(* Init ST08_407_B55_3 Hubtüre 4 Auslauf STN8 AST (ValveSensor) *)
ST08_407_B55_3.sInit.InstName            :='ST08_407_B55_3';
ST08_407_B55_3.sInit.BitName            :='+8_407_B55.3';
ST08_407_B55_3.sInit.Description         :='Hubtüre 4 Auslauf STN8 GST';
ST08_407_B55_3.sInit.SensorType          :=sValveSensorType_INIT;

(* Init ST08_408_B56_0 Rückhaltezylinder links Auslauf STN8 AST (ValveSensor) *)
ST08_408_B56_0.sInit.InstName            :='ST08_408_B56_0';
ST08_408_B56_0.sInit.BitName            :='+8_408_B56.0';
ST08_408_B56_0.sInit.Description         :='Rückhaltezylinder links Auslauf STN8 AST';
ST08_408_B56_0.sInit.SensorType          :=sValveSensorType_WORK;

(* Init ST08_408_B56_1 Rückhaltezylinder links Auslauf STN8 GST (ValveSensor) *)
ST08_408_B56_1.sInit.InstName            :='ST08_408_B56_1';
ST08_408_B56_1.sInit.BitName            :='+8_408_B56.1';
ST08_408_B56_1.sInit.Description         :='Rückhaltezylinder links Auslauf STN8 GST';
ST08_408_B56_1.sInit.SensorType          :=sValveSensorType_INIT;

(* Init ST08_408_B56_2 Rückhaltezylinder rechts Auslauf STN8 AST (ValveSensor) *)
ST08_408_B56_2.sInit.InstName            :='ST08_408_B56_2';
ST08_408_B56_2.sInit.BitName            :='+8_408_B56.2';
ST08_408_B56_2.sInit.Description         :='Rückhaltezylinder rechts Auslauf STN8 AST';
ST08_408_B56_2.sInit.SensorType          :=sValveSensorType_WORK;

(* Init ST08_408_B56_3 Rückhaltezylinder rechts Auslauf STN8 GST (ValveSensor) *)
ST08_408_B56_3.sInit.InstName            :='ST08_408_B56_3';
ST08_408_B56_3.sInit.BitName            :='+8_408_B56.3';
ST08_408_B56_3.sInit.Description         :='Rückhaltezylinder rechts Auslauf STN8 GST';
ST08_408_B56_3.sInit.SensorType          :=sValveSensorType_INIT;

(* Init ST08_408_B56_4 Abstapelzylinder 1 STN8 AST (ValveSensor) *)
ST08_408_B56_4.sInit.InstName            :='ST08_408_B56_4';
ST08_408_B56_4.sInit.BitName            :='+8_408_B56.4';
ST08_408_B56_4.sInit.Description         :='Abstapelzylinder 1 STN8 AST';
ST08_408_B56_4.sInit.SensorType          :=sValveSensorType_WORK;

(* Init ST08_408_B56_5 Abstapelzylinder 1 STN8 GST (ValveSensor) *)
ST08_408_B56_5.sInit.InstName            :='ST08_408_B56_5';
ST08_408_B56_5.sInit.BitName            :='+8_408_B56.5';
ST08_408_B56_5.sInit.Description         :='Abstapelzylinder 1 STN8 GST';
ST08_408_B56_5.sInit.SensorType          :=sValveSensorType_INIT;

(* Init ST08_408_B56_6 Abstapelzylinder 2 STN8 AST (ValveSensor) *)
ST08_408_B56_6.sInit.InstName            :='ST08_408_B56_6';
ST08_408_B56_6.sInit.BitName            :='+8_408_B56.6';
ST08_408_B56_6.sInit.Description         :='Abstapelzylinder 2 STN8 AST';
ST08_408_B56_6.sInit.SensorType          :=sValveSensorType_WORK;

(* Init ST08_408_B56_7 Abstapelzylinder 2 STN8 AST (ValveSensor) *)
ST08_408_B56_7.sInit.InstName            :='ST08_408_B56_7';
ST08_408_B56_7.sInit.BitName            :='+8_408_B56.7';
ST08_408_B56_7.sInit.Description         :='Abstapelzylinder 2 STN8 GST';
ST08_408_B56_7.sInit.SensorType          :=sValveSensorType_INIT;

(*ST08_400_B50_1 Stopper links + rechts Traystapel Auslaufband eingefahren (ValveSensor)*)
ST08_400_B50_1.sInit.InstName            :='ST08_400_B50_1';
ST08_400_B50_1.sInit.BitName            :='+8_400_B50.1';
ST08_400_B50_1.sInit.Description         :='Stopper links + rechts Auslauf STN8 AST';
ST08_400_B50_1.sInit.SensorType          :=sValveSensorType_WORK;

(*ST08_400_B50_2 Stopper links + rechts Traystapel Auslaufband ausgefahren (ValveSensor)*)
ST08_400_B50_2.sInit.InstName            :='ST08_400_B50_2';
ST08_400_B50_2.sInit.BitName            :='+8_400_B50.2';
ST08_400_B50_2.sInit.Description         :='Stopper links + rechts Auslauf STN8 GST';
ST08_400_B50_2.sInit.SensorType          :=sValveSensorType_INIT;

(*ST08_400_B50_3 Stopper links + rechts Traystapel Auslaufband eingefahren (ValveSensor)*)
ST08_400_B50_3.sInit.InstName            :='ST08_400_B50_3';
ST08_400_B50_3.sInit.BitName            :='+8_400_B50.3';
ST08_400_B50_3.sInit.Description         :='Stopper links + rechts Auslauf STN8 AST';
ST08_400_B50_3.sInit.SensorType          :=sValveSensorType_WORK;

(*ST08_400_B50_6 Stopper links + rechts Traystapel Auslaufband ausgefahren (ValveSensor)*)
ST08_400_B50_6.sInit.InstName            :='ST08_400_B50_6';
ST08_400_B50_6.sInit.BitName            :='+8_400_B50.6';
ST08_400_B50_6.sInit.Description         :='Stopper links + rechts Auslauf STN8 GST';
ST08_400_B50_6.sInit.SensorType          :=sValveSensorType_INIT;

(*ST08_401_B50_7 Traystapel schieben hinten ausgefahren (ValveSensor)*)
ST08_401_B50_7.sInit.InstName            :='ST08_401_B50_7';
ST08_401_B50_7.sInit.BitName            :='+8_401_B50.7';
ST08_401_B50_7.sInit.Description         :='Traystapel schieben hinten';
ST08_401_B50_7.sInit.SensorType          :=sValveSensorType_INIT;

(*ST08_412_B58_0 Rüstsatz Förderband Vereinzelner ausgefahren (ValveSensor)*)
ST08_412_B58_0.sInit.InstName            :='ST08_412_B58_0';
ST08_412_B58_0.sInit.BitName          	 :='+8_412_B58.0';
ST08_412_B58_0.sInit.Description         :='Rüstsatz Förderband Vereinzelner STN8 AST';
ST08_412_B58_0.sInit.SensorType          :=sValveSensorType_WORK;

(*ST08_412_B58_1 Rüstsatz Förderband Vereinzelner eingefahren (ValveSensor)*)
ST08_412_B58_1.sInit.InstName            :='ST08_412_B58_1';
ST08_412_B58_1.sInit.BitName          	 :='+8_412_B58.1';
ST08_412_B58_1.sInit.Description         :='Rüstsatz Förderband Vereinzelner STN8 GST';
ST08_412_B58_1.sInit.SensorType          :=sValveSensorType_INIT;

(*ST08_412_B58_2 Rüstsatz Förderband Stopper ausgefahren (ValveSensor)*)
ST08_412_B58_2.sInit.InstName            :='ST08_412_B58_2';
ST08_412_B58_2.sInit.BitName           	 :='+8_412_B58.2';
ST08_412_B58_2.sInit.Description         :='Rüstsatz Förderband Stopper STN8 AST';
ST08_412_B58_2.sInit.SensorType          :=sValveSensorType_WORK;

(*ST08_412_B58_3 Rüstsatz Förderband Stopper eingefahren (ValveSensor)*)
ST08_412_B58_3.sInit.InstName            :='ST08_412_B58_3';
ST08_412_B58_3.sInit.BitName            :='+8_412_B58.3';
ST08_412_B58_3.sInit.Description         :='Rüstsatz Förderband Stopper STN8 GST';
ST08_412_B58_3.sInit.SensorType          :=sValveSensorType_INIT;

(* Init ST08_412_B58_4 Rüstsatz Förderband frei zum Ablegen ISK von SP Maschine Position 1 (DigIn) *)
ST08_412_B58_4.sInit.InstName            :='ST08_412_B58_4';
ST08_412_B58_4.sInit.Description         :='Frei SP Maschine Position 1';
ST08_412_B58_4.sInit.BitInName           :='+8-412_B58.4';
ST08_412_B58_4.sInit.HomePosSignal       :=2; (* 0: Signal=Low, 1: Signal=High, 2: always  *)
ST08_412_B58_4.sInit.MaxTime             :=2000;

(* Init ST08_412_B58_5 Rüstsatz Förderband frei zum Ablegen ISK von SP Maschine Position 2 (DigIn) *)
ST08_412_B58_5.sInit.InstName            :='ST08_412_B58_5';
ST08_412_B58_5.sInit.Description         :='Frei SP Maschine Position 2';
ST08_412_B58_5.sInit.BitInName           :='+8-412_B58.5';
ST08_412_B58_5.sInit.HomePosSignal       :=2; (* 0: Signal=Low, 1: Signal=High, 2: always  *)
ST08_412_B58_5.sInit.MaxTime             :=2000;

(* Init ST08_412_B58_6 Rüstsatz Förderband frei zum Ablegen ISK von SP Maschine Position 3 (DigIn) *)
ST08_412_B58_6.sInit.InstName            :='ST08_412_B58_6';
ST08_412_B58_6.sInit.Description         :='Frei SP Maschine Position 3';
ST08_412_B58_6.sInit.BitInName           :='+8-412_B58.6';
ST08_412_B58_6.sInit.HomePosSignal       :=2; (* 0: Signal=Low, 1: Signal=High, 2: always  *)
ST08_412_B58_6.sInit.MaxTime             :=2000;

(* Init ST08_412_B58_5_35pol Lageerkennung links (DigIn) *)
ST08_412_B58_5_35pol.sInit.InstName            :='ST08_412_B58_5_35pol';
ST08_412_B58_5_35pol.sInit.Description         :=' Lageerkennung rechts';
ST08_412_B58_5_35pol.sInit.BitInName           :='+8-412_B58.5';
ST08_412_B58_5_35pol.sInit.HomePosSignal       :=2; (* 0: Signal=Low, 1: Signal=High, 2: always  *)
ST08_412_B58_5_35pol.sInit.MaxTime             :=2000;

(* Init ST08_412_B58_6_35pol Lageerkennung rechts (DigIn) *)
ST08_412_B58_6_35pol.sInit.InstName            :='ST08_412_B58_6_35pol';
ST08_412_B58_6_35pol.sInit.Description         :=' Lageerkennung links';
ST08_412_B58_6_35pol.sInit.BitInName           :='+8-412_B58.6';
ST08_412_B58_6_35pol.sInit.HomePosSignal    :=2; (* 0: Signal=Low, 1: Signal=High, 2: always  *)
ST08_412_B58_6_35pol.sInit.MaxTime             :=2000;

(* Init ST08_412_B58_7 Rüstsatz Förderband ISK anwesend zum Vereinzeln (DigIn) *)
ST08_412_B58_7.sInit.InstName            :='ST08_412_B58_7';
ST08_412_B58_7.sInit.Description         :='ISK anwesend zum Vereinzeln';
ST08_412_B58_7.sInit.BitInName           :='+8-412_B58.7';
ST08_412_B58_7.sInit.HomePosSignal       :=2; (* 0: Signal=Low, 1: Signal=High, 2: always  *)
ST08_412_B58_7.sInit.MaxTime             :=2000;

(* Init ST08_412_B59_0 Rüstsatz Förderband ISK auf Übergabeposition Roboter Verpackung (DigIn) *)
ST08_412_B59_0.sInit.InstName            :='ST08_412_B59_0';
ST08_412_B59_0.sInit.Description         :='ISK auf Übergabeposition Roboter';
ST08_412_B59_0.sInit.BitInName           :='+8-412_B59.0';
ST08_412_B59_0.sInit.HomePosSignal       :=2; (* 0: Signal=Low, 1: Signal=High, 2: always  *)
ST08_412_B59_0.sInit.MaxTime             :=2000;

(* Init ST08_169_K1 Bandantrieb 1 Einlauf Trays Ein (DigOutIn) *)
ST08_169_K1.sInit.InstName               :='ST08_169_K1';
ST08_169_K1.sInit.Description            :='Bandantrieb 1 Einlauf Trays Ein';
ST08_169_K1.sInit.BitOutName             :='+8-169_K1'; 
ST08_169_K1.sInit.BitInName              :='';
ST08_169_K1.sInit.HomePosOutput          :=2; (* 0: Signal=Low, 1: Signal=High, 2: always  *)
ST08_169_K1.sInit.MaxTime                :=2000;
ST08_169_K1.sInit.EnableInEveryMode  :=TRUE;

(* Init ST08_169_K2 Bandantrieb 4 Auslauf leere Trays Ein (DigOutIn) *)
ST08_169_K2.sInit.InstName               :='ST08_169_K2';
ST08_169_K2.sInit.Description            :='Bandantrieb 4 Auslauf leere Trays Ein';
ST08_169_K2.sInit.BitOutName             :='+8-169_K2'; 
ST08_169_K2.sInit.BitInName              :='';
ST08_169_K2.sInit.HomePosOutput          :=2; (* 0: Signal=Low, 1: Signal=High, 2: always  *)
ST08_169_K2.sInit.MaxTime                :=2000;
ST08_169_K2.sInit.EnableInEveryMode  :=TRUE;

(* Init ST08_170_K1 Bandantrieb 2 Hubquereinheit Trays Ein (DigOutIn) *) 
ST08_170_K1.sInit.InstName               :='ST08_170_K1';
ST08_170_K1.sInit.Description            :='Bandantrieb 2 Hubquereinheit Trays Ein';
ST08_170_K1.sInit.BitOutName             :='+8-170_K1';
ST08_170_K1.sInit.BitInName              :='';
ST08_170_K1.sInit.HomePosOutput          :=2; (* 0: Signal=Low, 1: Signal=High, 2: always  *)
ST08_170_K1.sInit.MaxTime                :=2000;
ST08_170_K1.sInit.EnableInEveryMode  :=TRUE;

(* Init ST08_170_K2 Bandantrieb 3 Hubquereinheit Trays Ein (DigOutIn) *)
ST08_170_K2.sInit.InstName               :='ST08_170_K2';
ST08_170_K2.sInit.Description            :='Bandantrieb 3 Hubquereinheit Trays Ein';
ST08_170_K2.sInit.BitOutName             :='+8-170_K2';
ST08_170_K2.sInit.BitInName              :='';
ST08_170_K2.sInit.HomePosOutput          :=2; (* 0: Signal=Low, 1: Signal=High, 2: always  *)
ST08_170_K2.sInit.MaxTime                :=2000;
ST08_170_K2.sInit.EnableInEveryMode  :=TRUE;

(* Init ST08_400_Y50_0 Stopper Traystapel Einlaufb. hinten links + rechts AST (Valve) *)
ST08_400_Y50_0.sInit.InstName            :='ST08_400_Y50_0';
ST08_400_Y50_0.sInit.BitName            :='+8-400_Y50.0';
ST08_400_Y50_0.sInit.Description         :='Stopper Traystapel Einlaufb. hinten links + rechts AST';
ST08_400_Y50_0.sInit.HomePosDefine       :=HOME_INIT;
ST08_400_Y50_0.sInit.InitDescription     :='GS ausfahren';
ST08_400_Y50_0.sInit.WorkDescription     :='AS einfahren';
ST08_400_Y50_0.sInit.DampBothTime        :=200;
ST08_400_Y50_0.sInit.KindOfValve         :='2G';
ST08_400_Y50_0.sInit.MaxTime             :=2000;

(* Init ST08_400_Y50_2 Stopper Traystapel Einlaufb. mitte links + rechts AST (Valve) *)
ST08_400_Y50_2.sInit.InstName            :='ST08_400_Y50_2';
ST08_400_Y50_2.sInit.BitName            :='+8-400_Y50.2';
ST08_400_Y50_2.sInit.Description         :='Stopper Traystapel Einlaufb. mitte links + rechts AST';
ST08_400_Y50_2.sInit.HomePosDefine       :=HOME_INIT;
ST08_400_Y50_2.sInit.InitDescription     :='GS ausfahren';
ST08_400_Y50_2.sInit.WorkDescription     :='AS einfahren';
ST08_400_Y50_2.sInit.DampBothTime        :=200;
ST08_400_Y50_2.sInit.KindOfValve         :='2G';
ST08_400_Y50_2.sInit.MaxTime             :=2000;

(* Init ST08_402_Y50_4 Stopper Traystapel Einlaufb. vorne links + rechts AST (Valve) *) 
ST08_402_Y50_4.sInit.InstName            :='ST08_402_Y50_4';
ST08_402_Y50_4.sInit.BitName            :='+8-402_Y50.4';
ST08_402_Y50_4.sInit.Description         :='Stopper Traystapel Einlaufb. vorne links + rechts AST';
ST08_402_Y50_4.sInit.HomePosDefine       :=HOME_INIT;
ST08_402_Y50_4.sInit.InitDescription     :='GS ausfahren';
ST08_402_Y50_4.sInit.WorkDescription     :='AS einfahren';
ST08_402_Y50_4.sInit.DampBothTime        :=200;
ST08_402_Y50_4.sInit.KindOfValve         :='2G';
ST08_402_Y50_4.sInit.MaxTime             :=2000;

(* Init ST08_403_Y50_6 Vakuum 1 Einlauf STN8 AST (Valve) *)
ST08_403_Y50_6.sInit.InstName            :='ST08_403_Y50_6';
ST08_403_Y50_6.sInit.BitName            :='+8-403_Y50.6';
ST08_403_Y50_6.sInit.Description         :='Vakuum 1 Einlauf STN8 AST';
ST08_403_Y50_6.sInit.HomePosDefine       :=HOME_ALWAYS;
ST08_403_Y50_6.sInit.InitDescription     :='OFF';
ST08_403_Y50_6.sInit.WorkDescription     :='ON';
ST08_403_Y50_6.sInit.DampBothTime        :=0;
ST08_403_Y50_6.sInit.KindOfValve         :='A';
ST08_403_Y50_6.sInit.MaxTime             :=2000;

(* Init ST08_403_Y50_7 Vakuum 2 Einlauf STN8 AST (Valve) *)
ST08_403_Y50_7.sInit.InstName            :='ST08_403_Y50_7';
ST08_403_Y50_7.sInit.BitName            :='+8-403_Y50.7';
ST08_403_Y50_7.sInit.Description         :='Vakuum 2 Einlauf STN8 AST';
ST08_403_Y50_7.sInit.HomePosDefine       :=HOME_ALWAYS;
ST08_403_Y50_7.sInit.InitDescription     :='OFF';
ST08_403_Y50_7.sInit.WorkDescription     :='ON';
ST08_403_Y50_7.sInit.DampBothTime        :=0;
ST08_403_Y50_7.sInit.KindOfValve         :='A';
ST08_403_Y50_7.sInit.MaxTime             :=2000;

(* Init ST08_405_Y51_0 Hubtüre 2 Einlauf Isokörper STN8 AST (Valve) *)
ST08_405_Y51_0.sInit.InstName            :='ST08_405_Y51_0';
ST08_405_Y51_0.sInit.BitName            :='+8-405_Y51.0';
ST08_405_Y51_0.sInit.Description         :='Hubtüre 2 Einlauf Isokörper STN8 AST';
ST08_405_Y51_0.sInit.HomePosDefine       :=HOME_INIT;
ST08_405_Y51_0.sInit.InitDescription     :='GS ausfahren';
ST08_405_Y51_0.sInit.WorkDescription     :='AS einfahren';
ST08_405_Y51_0.sInit.DampBothTime        :=0;
ST08_405_Y51_0.sInit.KindOfValve         :='2G';
ST08_405_Y51_0.sInit.MaxTime             :=5000;

(* Init ST08_406_Y51_2 Hubtüre 3 STN8 AST (Valve) *)
ST08_406_Y51_2.sInit.InstName            :='ST08_406_Y51_2';
ST08_406_Y51_2.sInit.BitName            :='+8-406_Y51.2';
ST08_406_Y51_2.sInit.Description         :='Hubtüre 3 Auslauf STN8 AST';
ST08_406_Y51_2.sInit.HomePosDefine       :=HOME_INIT;
ST08_406_Y51_2.sInit.InitDescription     :='GS ausfahren';
ST08_406_Y51_2.sInit.WorkDescription     :='AS einfahren';
ST08_406_Y51_2.sInit.DampBothTime        :=0;
ST08_406_Y51_2.sInit.KindOfValve         :='2G';
ST08_406_Y51_2.sInit.MaxTime             :=5000;

(* Init ST08_407_Y51_4 Hubtüre 4 Auslauf STN8 AST (Valve) *)
ST08_407_Y51_4.sInit.InstName            :='ST08_407_Y51_4';
ST08_407_Y51_4.sInit.BitName            :='+8-407_Y51.4';
ST08_407_Y51_4.sInit.Description         :='Hubtüre 4 Auslauf STN8 AST';
ST08_407_Y51_4.sInit.HomePosDefine       :=HOME_ALWAYS;
ST08_407_Y51_4.sInit.InitDescription     :='GS ausfahren';
ST08_407_Y51_4.sInit.WorkDescription     :='AS einfahren';
ST08_407_Y51_4.sInit.DampBothTime        :=0;
ST08_407_Y51_4.sInit.KindOfValve         :='2G';
ST08_407_Y51_4.sInit.MaxTime             :=10000;

(* Init ST08_404_Y51_6 Stopper Traystapel Isokörper AST (Valve) *)
ST08_404_Y51_6.sInit.InstName            :='ST08_404_Y51_6';
ST08_404_Y51_6.sInit.BitName            :='+8-404_Y51.6';
ST08_404_Y51_6.sInit.Description         :='Stopper Traystapel Isokörper AST';
ST08_404_Y51_6.sInit.HomePosDefine       :=HOME_INIT;
ST08_404_Y51_6.sInit.InitDescription     :='GS ausfahren';
ST08_404_Y51_6.sInit.WorkDescription     :='AS einfahren';
ST08_404_Y51_6.sInit.DampBothTime        :=200;
ST08_404_Y51_6.sInit.KindOfValve         :='2G';
ST08_404_Y51_6.sInit.MaxTime             :=2000;

(* Init ST08_404_Y52_0 Hub Bandstrecke STN8 AST (Valve) *)
ST08_404_Y52_0.sInit.InstName            :='ST08_404_Y52_0';
ST08_404_Y52_0.sInit.BitName            :='+8-404_Y52.0';
ST08_404_Y52_0.sInit.Description         :='Hub Bandstrecke STN8 AST';
ST08_404_Y52_0.sInit.HomePosDefine       :=HOME_INIT;
ST08_404_Y52_0.sInit.InitDescription     :='GS einfahren';
ST08_404_Y52_0.sInit.WorkDescription     :='AS ausfahren';
ST08_404_Y52_0.sInit.DampBothTime        :=200;
ST08_404_Y52_0.sInit.KindOfValve         :='2G';
ST08_404_Y52_0.sInit.MaxTime             :=2000;


(* Init ST08_406_Y52_3 Ausheber Trays Entnahmepos. Isok. STN8 GST (Valve) *)
ST08_406_Y52_3.sInit.InstName            :='ST08_406_Y52_3';
ST08_406_Y52_3.sInit.BitName            :='+8-406_Y52.3';
ST08_406_Y52_3.sInit.Description         :='Ausheber Trays Entnahmepos. Isok. STN8 GST';
ST08_406_Y52_3.sInit.HomePosDefine       :=HOME_ALWAYS;
ST08_406_Y52_3.sInit.InitDescription     :='GS einfahren';
ST08_406_Y52_3.sInit.WorkDescription     :='AS ausfahren';
ST08_406_Y52_3.sInit.DampBothTime        :=200;
ST08_406_Y52_3.sInit.KindOfValve         :='2G';
ST08_406_Y52_3.sInit.MaxTime             :=3000;

(* Init ST08_401_Y52_4 Traystapel schieben hinten AST (Valve) *)
ST08_401_Y52_4.sInit.InstName            :='ST08_401_Y52_4';
ST08_401_Y52_4.sInit.BitName            :='+8-401_Y52.4';
ST08_401_Y52_4.sInit.Description         :='Traystapel schieben hinten';
ST08_401_Y52_4.sInit.HomePosDefine       :=HOME_INIT;
ST08_401_Y52_4.sInit.InitDescription     :='GS einfahren';
ST08_401_Y52_4.sInit.WorkDescription     :='AS ausfahren';
ST08_401_Y52_4.sInit.DampBothTime        :=200;
ST08_401_Y52_4.sInit.KindOfValve         :='2G';
ST08_401_Y52_4.sInit.MaxTime             :=2000;

(* Stopper links + rechts Traystapel Auslaufband einfahren (Valve) *)
ST08_400_Y52_5.sInit.InstName            :='ST08_400_Y52_5';
ST08_400_Y52_5.sInit.BitName            :='+8-400_Y52.5';
ST08_400_Y52_5.sInit.Description         :='Stopperzylinder li+re STN8 AST';
ST08_400_Y52_5.sInit.HomePosDefine       :=HOME_BOTH;
ST08_400_Y52_5.sInit.InitDescription     :='GS ausfahren';
ST08_400_Y52_5.sInit.WorkDescription     :='AS einfahren';
ST08_400_Y52_5.sInit.DampBothTime        :=200;
ST08_400_Y52_5.sInit.KindOfValve         :='2G';
ST08_400_Y52_5.sInit.MaxTime             :=3000;

(* Init ST08_402_Y52_6 Traystapel schieben mitte AST (Valve) *)
ST08_402_Y52_6.sInit.InstName            :='ST08_402_Y52_6';
ST08_402_Y52_6.sInit.BitName            :='+8-402_Y52.6';
ST08_402_Y52_6.sInit.Description         :='Traystapel schieben mitte';
ST08_402_Y52_6.sInit.HomePosDefine       :=HOME_INIT;
ST08_402_Y52_6.sInit.InitDescription     :='GS einfahren';
ST08_402_Y52_6.sInit.WorkDescription     :='AS ausfahren';
ST08_402_Y52_6.sInit.DampBothTime        :=200;
ST08_402_Y52_6.sInit.KindOfValve         :='2G';
ST08_402_Y52_6.sInit.MaxTime             :=2000;

(* Init ST08_402_Y52_7 Traystapel schieben vorne AST (Valve) *)
ST08_402_Y52_7.sInit.InstName            :='ST08_402_Y52_7';
ST08_402_Y52_7.sInit.BitName            :='+8-402_Y52.7';
ST08_402_Y52_7.sInit.Description         :='Traystapel schieben vorne';
ST08_402_Y52_7.sInit.HomePosDefine       :=HOME_INIT;
ST08_402_Y52_7.sInit.InitDescription     :='GS einfahren';
ST08_402_Y52_7.sInit.WorkDescription     :='AS ausfahren';
ST08_402_Y52_7.sInit.DampBothTime        :=200;
ST08_402_Y52_7.sInit.KindOfValve         :='2G';
ST08_402_Y52_7.sInit.MaxTime             :=2000;

(* Init ST08_404_Y53_0 Abstapelzylinder 1 AST (Valve) *)
ST08_404_Y53_0.sInit.InstName            :='ST08_404_Y53_0';
ST08_404_Y53_0.sInit.BitName            :='+8-404_Y53.0';
ST08_404_Y53_0.sInit.Description         :='Abstapelzylinder 1 AST';
ST08_404_Y53_0.sInit.HomePosDefine       :=HOME_INIT;
ST08_404_Y53_0.sInit.InitDescription     :='GS einfahren';
ST08_404_Y53_0.sInit.WorkDescription     :='AS ausfahren';
ST08_404_Y53_0.sInit.DampBothTime        :=400;
ST08_404_Y53_0.sInit.KindOfValve         :='2G';
ST08_404_Y53_0.sInit.MaxTime             :=3000;

(* Init ST08_404_Y53_2 Abstapelzylinder 2  AST (Valve) *)
ST08_404_Y53_2.sInit.InstName            :='ST08_404_Y53_2';
ST08_404_Y53_2.sInit.BitName            :='+8-404_Y53.2';
ST08_404_Y53_2.sInit.Description         :='Abstapelzylinder 2  AST';
ST08_404_Y53_2.sInit.HomePosDefine       :=HOME_INIT;
ST08_404_Y53_2.sInit.InitDescription     :='GS einfahren';
ST08_404_Y53_2.sInit.WorkDescription     :='AS ausfahren';
ST08_404_Y53_2.sInit.DampBothTime        :=200;
ST08_404_Y53_2.sInit.KindOfValve         :='2G';
ST08_404_Y53_2.sInit.MaxTime             :=3000;

(* Init ST08_405_Y53_4 Rückhaltezylinder li+re Traystapel Isokörper AST (Valve) *) 
ST08_405_Y53_4.sInit.InstName            :='ST08_405_Y53_4';
ST08_405_Y53_4.sInit.BitName            :='+8-405_Y53.4';
ST08_405_Y53_4.sInit.Description         :='Rückhaltezylinder li+re Traystapel Isokörper AST';
ST08_405_Y53_4.sInit.HomePosDefine       :=HOME_ALWAYS;
ST08_405_Y53_4.sInit.InitDescription     :='GS einfahren';
ST08_405_Y53_4.sInit.WorkDescription     :='AS ausfahren';
ST08_405_Y53_4.sInit.DampBothTime        :=200;
ST08_405_Y53_4.sInit.KindOfValve         :='2G';
ST08_405_Y53_4.sInit.MaxTime             :=3000;

(* Init ST08_408_Y54_0 Rückhaltezylinder li.+re. Auslauf STN8 AST (Valve) *)
ST08_408_Y54_0.sInit.InstName            :='ST08_408_Y54_0';
ST08_408_Y54_0.sInit.BitName            :='+8-408_Y54.0';
ST08_408_Y54_0.sInit.Description         :='Rückhaltezylinder li.+re. Auslauf STN8 AST';
ST08_408_Y54_0.sInit.HomePosDefine       :=HOME_INIT;(*HOME_ALWAYS;*)
ST08_408_Y54_0.sInit.InitDescription     :='GS einfahren';
ST08_408_Y54_0.sInit.WorkDescription     :='AS ausfahren';
ST08_408_Y54_0.sInit.DampBothTime        :=200;
ST08_408_Y54_0.sInit.KindOfValve         :='2G';
ST08_408_Y54_0.sInit.MaxTime             :=3000;

(* Init ST08_408_Y54_2 Abstapelzylinder 1 STN8 AST (Valve) *)
ST08_408_Y54_2.sInit.InstName            :='ST08_408_Y54_2';
ST08_408_Y54_2.sInit.BitName            :='+8-408_Y54.2';
ST08_408_Y54_2.sInit.Description         :='Aufstapelzylinder 1 STN8 AST';
ST08_408_Y54_2.sInit.HomePosDefine       :=HOME_INIT;
ST08_408_Y54_2.sInit.InitDescription     :='GS einfahren';
ST08_408_Y54_2.sInit.WorkDescription     :='AS ausfahren';
ST08_408_Y54_2.sInit.DampBothTime        :=200;
ST08_408_Y54_2.sInit.KindOfValve         :='2G';
ST08_408_Y54_2.sInit.MaxTime             :=3000;

(* Init ST08_408_Y54_4 Abstapelzylinder 2 STN8 AST (Valve) *)
ST08_408_Y54_4.sInit.InstName            :='ST08_408_Y54_4';
ST08_408_Y54_4.sInit.BitName            :='+8-408_Y54.4';
ST08_408_Y54_4.sInit.Description         :='Aufstapelzylinder 2 STN8 AST';
ST08_408_Y54_4.sInit.HomePosDefine       :=HOME_INIT;
ST08_408_Y54_4.sInit.InitDescription     :='GS einfahren';
ST08_408_Y54_4.sInit.WorkDescription     :='AS ausfahren';
ST08_408_Y54_4.sInit.DampBothTime        :=200;
ST08_408_Y54_4.sInit.KindOfValve         :='2G';
ST08_408_Y54_4.sInit.MaxTime             :=3000;

(* Rüstsatz Förderband Vereinzelner (Valve) *)
ST08_412_Y55_0.sInit.InstName            :='ST08_412_Y55_0';
ST08_412_Y55_0.sInit.BitName            :='+8-412_Y55.0';
ST08_412_Y55_0.sInit.Description         :='Rüstsatz Förderband Vereinzelner';
ST08_412_Y55_0.sInit.HomePosDefine       :=HOME_ALWAYS;
ST08_412_Y55_0.sInit.InitDescription     :='GS einfahren';
ST08_412_Y55_0.sInit.WorkDescription     :='AS ausfahren';
ST08_412_Y55_0.sInit.DampBothTime        :=200;
ST08_412_Y55_0.sInit.KindOfValve         :='2G';
ST08_412_Y55_0.sInit.MaxTime             :=3000;

(* Rüstsatz Förderband Stopper (Valve) *)
ST08_412_Y55_2.sInit.InstName            :='ST08_412_Y55_2';
ST08_412_Y55_2.sInit.BitName            :='+8-412_Y55.2';
ST08_412_Y55_2.sInit.Description         :='Rüstsatz Förderband Stopper';
ST08_412_Y55_2.sInit.HomePosDefine       :=HOME_ALWAYS;
ST08_412_Y55_2.sInit.InitDescription     :='GS einfahren';
ST08_412_Y55_2.sInit.WorkDescription     :='AS ausfahren';
ST08_412_Y55_2.sInit.DampBothTime        :=200;
ST08_412_Y55_2.sInit.KindOfValve         :='2G';
ST08_412_Y55_2.sInit.MaxTime             :=3000;
END_PROGRAM

(* POU Stations/ST_03_Ruestsaetze/ST_03_PRGs/ST03_Band_alt, ST *)
PROGRAM ST03_Band_alt
VAR_INPUT
	b_MoveRel 		:BOOL;
	fb_ton_Stopp_Band					: TON;
	bLockBand : BOOL;
END_VAR
VAR
	b_PosBetrieb	:BOOL;
	fb_rTrig_Off		: R_TRIG;
	fb_rTrig_stop		: R_TRIG;
	fb_ton_Off			: TON;
	fb_ton_Off2			: TON;
	fb_rTrig_On			: R_TRIG;
	fb_ton_Stau			: TON;
	fb_ton_Stau2		: TON;
	fb_rtrig_Stopp_Band	: R_TRIG;

	fb_rTrig_MoveRel	: R_TRIG;

	MsgOK				: BOOL;
	MsgCancel			: BOOL;
	lr_PT				: LREAL;
END_VAR
fb_ton_Stopp_Band(IN:= ,PT:=t#10m , Q=> , ET=> );																	(*Stop Wenn von der Sritzguss kein Teile kommen*)

fb_rtrig_Stopp_Band(CLK:=ST00_72_X1_3.BitInToCheck OR ST02_FDB_80_B02.BitInToCheck);
IF	fb_rtrig_Stopp_Band.Q THEN
	fb_ton_Stopp_Band.IN:=FALSE;
END_IF

(*Störung Oriental Motor bei SG-Maschine 3621*)
IF MP.ST03.SGM_3621 THEN
	IF NOT St03_V2.BitInToCheck THEN
		ST03_A5.SetSignalLow := TRUE;

		MessageHandler.Msg.ID:='PM101';
		MessageHandler.Msg.Color:=Color.red;
		MessageHandler.Msg.Name:='Error Förderband';
		MessageHandler.Msg.Text:='Störung Motor Oriental Förderband!';
		MessageHandler.Msg.Station:=3;

		MessageHandler(
			Prio:=2, 							(*1=highest, .. , 4=lowest*)
			Btn1Addr:=ADR(MsgOk),				(*Address of Button1 , if Zero then Button is unvisible*)
			Btn2Addr:=0(*ADR(MsgCancel)*),		(*Address of Button2 , if Zero then Button is unvisible*)
			sVisu:=Visu.Message);
	END_IF
END_IF
(*Motorregelung einschalten=========================================================== *)

IF NOT MP.ST03.SGM_3621 THEN
	IF  NOT ST03_51_M1.Error_ THEN
		IF	(NOT Safety_Fuses_AirPressure.SafetyOK OR gRunEmpty) AND
			ST03_51_M1.on THEN
			ST03_51_M1.MotorOff :=TRUE;
		END_IF

		IF	ModeSelect.Mode > MODE_MANUAL AND
			NOT gRunEmpty AND
			Safety_Fuses_AirPressure.SafetyOK AND
			NOT ST03_51_M1.on THEN
			ST03_51_M1.MotorOn :=TRUE;
		END_IF
	END_IF
END_IF

(*Fahren bis zu Flügelkamera Förderband============================================================ *)

IF	gTypeCode=312  OR		(*93pol*)
	gTypeCode=4991 THEN	(*102pol*)
	b_PosBetrieb:=TRUE;
	(*Impolsbetrieb Förderband============================================================ *)

	IF 	ST03_IFM_Camera.State=STATE_WAIT OR
 		ModeSelect.Mode>=MODE_MANUAL OR
		NOT MP.ST00.IFMCameraActive THEN

		fb_rTrig_MoveRel(CLK:= ST03_51_M1.Ready AND
								b_MoveRel);

		IF	fb_rTrig_MoveRel.Q THEN
			ST03_51_M1.sVelo.maxRpm;
			ST03_51_M1.Vorgabe_Velo:=16000; 			(*mm/min*)
			ST03_51_M1.Vorgabe_Pos_Rel:=MP.ST02.IFMPos;
			ST03_51_M1.MoveRel:=TRUE;
		END_IF

	END_IF

ELSE
	(*Dauerbetrieb Förderband============================================================ *)
	b_PosBetrieb:=FALSE;
	fb_ton_Off(IN:=ST00_73_K3.BitOutToSet , PT:=t#5m, Q=> , ET=> );			(*Stop Wenn von der SG-Maschine keine Teile kommen*)

	IF  gTypeCode = 322 THEN (*160pol*)
		fb_ton_Off2(IN:=ST00_73_K3.BitOutToSet AND								(* Schnittstelle Förderband frei für Spritzmaschine*)
						ST03_422_B64_4.BitInToCheck AND						(* Teil auf Abholposition Roboter *)
						(Robot01.ActualArea<>4), PT:=t#5s , Q=> , ET=> ); 			(*anhalten wenn Roboter nicht in der WT Area ist, die Ablageposition leer und die Abholposition voll ist*)
	ELSE
		fb_ton_Off2(IN:=ST00_73_K3.BitOutToSet AND								(* Schnittstelle Förderband frei für Spritzmaschine*)
						ST08_412_B59_0.BitInToCheck AND						(* Teil auf Abholposition Roboter *)
						(Robot01.ActualArea<>4), PT:=t#3s , Q=> , ET=> ); 		(*anhalten wenn Roboter nicht in der WT Area ist, die Ablageposition leer und die Abholposition voll ist*)
	END_IF

	IF gTypeCode = 5841 THEN	(*268pol*)
		(*Stop wenn 4 Teile auf unterer Führungsschiene belegt sind *)
		fb_ton_Stau2(IN:=	ModeSelect.Mode > MODE_MANUAL AND
							ST03_556_B69_5.BitInToCheck AND	(* Führungsschiene Überwachung Staustrecke*)
							(ST03_556_B69_7. BitInToCheck OR	(* ISK anwesend an Abholposition*)
							Robot01.ActualArea <> 0	AND		(* Roboter zw. Abhol- und Park-Pos.*)
							Robot01.ActualArea <> 5 	AND		(* Blister Pos*)
							Robot01.ActualArea <> 6	), 			(* Park-Pos.*)
							PT:=t#500ms , Q=> , ET=> );
	ELSE
		IF  MP.ST03.SGM_3621 THEN
			fb_ton_Stau.PT:=t#15s;
		ELSE
			lr_PT:=(112-MP.ST02.Override_Band) *0.25;
			fb_ton_Stau.PT:=LREAL_TO_TIME(lr_PT * 1000);
		END_IF
	
		fb_ton_Stau(IN:=	NOT ST00_73_K3.BitOutToSet AND
							Robot01.ActualArea <> 4 AND
							(ModeSelect.Mode = MODE_AUTO_RUN OR ModeSelect.Mode = MODE_AUTO_STOP) ,
							Q=> , ET=>); 			(*Stop wenn Teile nach dem Ablegen nicht weiter gefördert werden*)
	END_IF

	fb_rTrig_Off(CLK:= ModeSelect.Mode<=MODE_MANUAL );

	fb_rTrig_stop(CLK:= ModeSelect.Mode<=MODE_MANUAL AND ST03_51_M1.sVisuAxis.BtnStop.Pressed );

	fb_rTrig_On(CLK:= 	ModeSelect.Mode>MODE_MANUAL AND
						Safety_Fuses_AirPressure.SafetyOK );

	IF NOT MP.ST03.SGM_3621 THEN
		IF	fb_rTrig_On.Q THEN
			ST03_51_M1.MotorOn:=TRUE;
		END_IF

		IF	ST03_51_M1.On THEN
			ST03_51_M1.MoveP:=MP.ST03.BandMoveP;
			ST03_51_M1.MoveN:=NOT MP.ST03.BandMoveP;
		END_IF

		IF 	NOT DummyTest_160pol AND
			(fb_rTrig_Off.Q OR
			fb_ton_Off2.Q OR
			fb_ton_Off.Q OR
			fb_ton_Stau.Q OR
			fb_ton_Stau2.Q OR
			fb_rTrig_stop.Q OR
			bLockBand) THEN
			ST03_51_M1.MotorOn:=FALSE;
			ST03_51_M1.MotorOff:=TRUE;
			ST03_51_M1.MoveN:=FALSE;
			ST03_51_M1.MoveP:=FALSE;
		ELSIF
			DummyTest_160pol AND NOT SpecialMode06.startBand THEN
			ST03_51_M1.MotorOn:=FALSE;
			ST03_51_M1.MotorOff:=TRUE;
			ST03_51_M1.MoveN:=FALSE;
			ST03_51_M1.MoveP:=FALSE;
		END_IF
	ELSE

		(*Ansteuerung Oriental Motor bei SG-Maschine 3621*)

		IF	NOT Safety_Fuses_AirPressure.SafetyOK THEN
			ST03_A5.SetSignalLow:=TRUE;
			ST03_A5.SetSignalHigh :=FALSE;
		ELSIF
			fb_rTrig_Off.Q OR fb_ton_Off2.Q OR fb_ton_Stau.Q THEN
			ST03_A5.SetSignalLow := TRUE;
			ST03_A5.SetSignalHigh :=FALSE;
		ELSIF
			ModeSelect.Mode >MODE_MANUAL AND
			Safety_Fuses_AirPressure.SafetyOK THEN
			ST03_A5.SetSignalHigh :=TRUE;
			ST03_A5.SetSignalLow := FALSE;
		END_IF
	END_IF


END_IF
END_PROGRAM

(* POU zLibrary/ept/Sprache/ST_SwitchLng, ST *)
PROGRAM ST_SwitchLng
VAR_OUTPUT
	b_EndChangeLng		: BOOL;
END_VAR
VAR
	fb_state_entry			: ST_StateEntry;
	s_sprache			: STRING(10);
	b_first_cycle			: BOOL := TRUE;

	btn_Language		: ARRAY [0..3] OF sButtonVisu;

	fbTon_ChangeLng		: TON;
END_VAR
VAR_TEMP
	i					:INT;
END_VAR
fbTon_ChangeLng(
	IN:=	ST_ReadXmlLineMsg.b_EndChangeLng AND
		ST_ReadXmlLine.b_EndChangeLng,
	PT:= t#200ms,
	Q=> b_EndChangeLng,
	ET=> );

IF 	b_first_cycle THEN
	IF	fb_state_entry.fb_ton_Step.ET > t#15s OR
		MP.ST00.Sprache <>'' THEN
		s_sprache := MP.ST00.Sprache;
		CURRENTLANGUAGE:=MP.ST00.Sprache;
		b_first_cycle := FALSE;
	END_IF
ELSE
	MP.ST00.Sprache := CURRENTLANGUAGE;
END_IF
Btn_Init();

IF		btn_Language[1].Pressed THEN
		CURRENTLANGUAGE:= 'DE';
ELSIF
		btn_Language[2].Pressed THEN
		CURRENTLANGUAGE:= 'EN';
ELSIF
		btn_Language[3].Pressed THEN
		CURRENTLANGUAGE:= 'CZ';
END_IF


(* ======================================Schrittkette======================================== *)
fb_state_entry(i16_pos:= 1);

CASE fb_state_entry.i16_step OF
(*=======================================================*)
	INIT_OBJ:

		fb_state_entry.i16_next_step := 10;

(*=======================================================*)
	INIT:
			;

END_CASE

fb_state_entry(i16_pos:= 2 );
END_PROGRAM
ACTION Btn_Init:
btn_Language[1].Text:='DE';
btn_Language[2].Text:='EN';
btn_Language[3].Text:='CZ';

FOR i := 0 TO 3  BY 1DO
	btn_Language[i].Enable:=TRUE;
	btn_Language[i].BackgroundColor:=Color.lightgrey;
	btn_Language[i].TextColor:=Color.black;
	btn_Language[i].Visible:= TRUE;

END_FOR


IF	CURRENTLANGUAGE = 'DE' THEN
	i:=1;
ELSIF
	CURRENTLANGUAGE = 'EN' THEN
	i:=2;
ELSIF
	CURRENTLANGUAGE = 'CZ' THEN
	i:=3;
ELSE
	i:=1;
END_IF

btn_Language[i].BackgroundColor:=Color.grey;
END_ACTION

(* POU zLibrary/ept/Checks/CheckBounds, ST *)
FUNCTION CheckBounds : DINT
VAR_INPUT
	index, lower, upper 	: DINT;
END_VAR
VAR
END_VAR
IF index<lower THEN
	CheckBounds_ErrCnt := CheckBounds_ErrCnt + 1;
	CheckBounds := lower;
ELSIF index>upper THEN
	CheckBounds_ErrCnt := CheckBounds_ErrCnt + 1;
	CheckBounds := upper;
ELSE
	CheckBounds := index;
END_IF
END_FUNCTION

(* POU zLibrary/ept/Checks/CheckDivByte, ST *)
FUNCTION CheckDivByte : BYTE
VAR_INPUT
	divisor			 	: BYTE;
END_VAR
VAR
END_VAR
IF divisor = 0 THEN
	CheckByteZeroDiv_ErrCnt := CheckByteZeroDiv_ErrCnt + 1;
	CheckDivByte := 1;
ELSE
	CheckDivByte := divisor;
END_IF
END_FUNCTION

(* POU zLibrary/ept/Checks/CheckDivDWord, ST *)
FUNCTION CheckDivDWord : DWORD
VAR_INPUT
	divisor				: DWORD;
END_VAR
VAR
END_VAR
IF divisor = 0 THEN
	CheckDWordZeroDiv_ErrCnt := CheckDWordZeroDiv_ErrCnt + 1;
	CheckDivDWord := 1;
ELSE
	CheckDivDWord := divisor;
END_IF
END_FUNCTION

(* POU zLibrary/ept/Checks/CheckDivReal, ST *)
FUNCTION CheckDivReal : REAL
VAR_INPUT
	divisor		 		: REAL;
END_VAR
VAR
END_VAR
IF divisor = 0 THEN
	CheckRealZeroDiv_ErrCnt := CheckRealZeroDiv_ErrCnt + 1;
	CheckDivReal := 1;
ELSE
	CheckDivReal := divisor;
END_IF
END_FUNCTION

(* POU zLibrary/ept/Checks/CheckDivWord, ST *)
FUNCTION CheckDivWord : WORD
VAR_INPUT
	divisor				: WORD;
END_VAR
VAR
END_VAR
IF divisor = 0 THEN
	CheckWordZeroDiv_ErrCnt:= CheckWordZeroDiv_ErrCnt + 1;
	CheckDivWord := 1;
ELSE
	CheckDivWord := divisor;
END_IF
END_FUNCTION

(* POU System/HelpFunctions/CheckProcTime, ST *)
FUNCTION_BLOCK CheckProcTime
VAR_OUTPUT
	PTime		: DINT;	(* Time since start of the timer *)
	Timeout		: BOOL; (* Flag if Timeout occured *)
END_VAR
VAR_INPUT
	MTime		: DINT;	(* Time to timeout *)
	Start		: BOOL;	(* True starts the Timer, False resets *)
END_VAR
VAR
	TONT		: TON;	(* Timer counting Timer *)
END_VAR
(* Start Timer if Start is True.
Stop Timer ,if Start is false.
Timer maximal counting to two hours. *)
TONT(IN:=Start,PT:=T#2h);

(* Updating the Processtime PTime. You get it if you change the output ET of TONT to DWORD.. *)
PTime:=TIME_TO_DWORD(TONT.ET);

(* Setting output Timeout
No Timeout IF Timer stopped OR mtime > ptime*)
IF 	MTime > PTime OR NOT Start THEN
	Timeout:=FALSE;
ELSE
	Timeout:=TRUE;
END_IF
END_FUNCTION_BLOCK

(* POU zLibrary/ept/Checks/CheckRangeSigned, ST *)
FUNCTION CheckRangeSigned : DINT
VAR_INPUT
    value, lower, upper: DINT;
END_VAR
VAR
END_VAR
IF (value < lower) THEN
	CheckRangeSigned_ErrCnt := CheckRangeSigned_ErrCnt + 1;
	CheckRangeSigned := lower;
ELSIF(value > upper) THEN
	CheckRangeSigned_ErrCnt := CheckRangeSigned_ErrCnt + 1;
	CheckRangeSigned := upper;
ELSE
	CheckRangeSigned := value;
END_IF
END_FUNCTION

(* POU zLibrary/ept/Checks/CheckRangeUnsigned, ST *)
FUNCTION CheckRangeUnsigned : UDINT
VAR_INPUT
    value, lower, upper: UDINT;
END_VAR
VAR
END_VAR
IF (value < lower) THEN
	CheckRangeUnSigned_ErrCnt := CheckRangeUnsigned_ErrCnt + 1;
	CheckRangeUnsigned := lower;
ELSIF(value > upper) THEN
	CheckRangeUnsigned_ErrCnt := CheckRangeUnsigned_ErrCnt + 1;
	CheckRangeUnsigned := upper;
ELSE
	CheckRangeUnsigned := value;
END_IF
END_FUNCTION

(* POU zLibrary/ept/Achse/fb_72x1_Achse, ST *)
FUNCTION_BLOCK fb_72x1_Achse   (*Coe-Online 7010.03 (CSV) velocity mode*)
VAR_INPUT
	Stop				:BOOL;			(*aktiven Verfahrbefehl beenden*)
	Reset				:BOOL;			(*Fehler quttieren*)
	MotorOn				:BOOL;			(*Regelung einschalten*)
	MotorOff			:BOOL;			(*Regelung abschalten*)
	NotausOK			:BOOL;
	Override			:DINT;
	Offset				:REAL;			(*  *)
	Vorgabe_Velo		:DINT;			(*in U/min oder mm/min*)
	MoveAbs				:BOOL;			(*startet Positionierung absolut*)
	MoveRel				:BOOL;			(*startet Positionierung relativ*)
	Vorgabe_Pos_Abs		:LREAL:=0;		(*auf diese Position wird bei start MoveAbs gefahren (mm oder Grad)*)
	Vorgabe_Pos_Rel		:LREAL:=0;		(*um diesen Wert wird die Achse bei start MoveRel gefahren (mm oder Grad)*)
	MoveP				:BOOL;			(*Achse bewegt sich in positiver Richtung solange MoveP TRUE ist, oder bis zum Softwarelimit*)
	MoveN				:BOOL;			(*Achse bewegt sich in negativer Richtung solange MoveN TRUE ist, oder bis zum Softwarelimit*)
	bMove				:BOOL;
	sConfig				:st_config_axis;	(*Initialisierung der Achse*)
	sPosList			:ARRAY [1..NO_OF_POS_AXIS] OF st_Pos;

	e_Position			AT %I* :UDINT;
	e_Statusword		AT %I* :UINT;
	e_Velocity			AT %I* :DINT;
	e_Torque			AT %I* :INT;
	e_Following_Error	AT %I* :DINT; 	(*Schleppfehler*)
	e_Toggle			AT %I* :BOOL;
	e_State				AT %I* :UINT;

END_VAR
VAR_OUTPUT
	a_Controlword		AT %Q* :UINT;
	a_Target_Velocity	AT %Q*: DINT;
	a_Target_Position	AT %Q* :UDINT;
	Torque				:ARRAY [1..NO_OF_Torque] OF INT;

	Busy				:BOOL;
	Done				:BOOL;		(*Achse steht auf Position*)
	Error_				:BOOL;
	Ready				:BOOL;
	On					:BOOL;		(*Motor in Regelung*)
	On_Position			:BOOL;		(*Achse steht auf Position*)
	Connect				:BOOL;		(*KLemme ist mit PLC verbunden*)
END_VAR
VAR_IN_OUT
	sVisu				:sDigInVisu;
END_VAR
VAR
	sHelp				:st_Help_axis;
	fb_state_entry		:ST_StateEntry;

	sFb					:st_fb_axis;

	sSm					:st_sm_axis;		(*Störmeldungen*)
	sSmEmpty			:st_sm_axis;
	sCtrl				:st_ctrl_Axis;		(*Control und Status*)
	sCtrlEmpty			:st_ctrl_Axis;

	sVisuAxis			:st_Visu_axis;		(*Taster der Visu*)
	sSdo				:st_sdo;

	(*Variablen für Behr Meldungen*)
	TempErrorText		:STRING(255);
	ProcessTime			:DINT;				(* Counts the time in steps of 100ms since starting operation *)
	Error				:ErrorStruct;
	LaufschriftErrh		:FB_Laufschrift;
	LaufschriftObj		:FB_Laufschrift;

	(*Regler*)
	sVelo				:st_Velo_axis;		(*Geschwindigkeiten*)
	sRegler				:st_PID_axis;		(*Var zur ermittling der Ausgabegeschwindigkeit*)
	sPos				:st_Pos_axis;		(*Positionen*)

	FB_ReadXmlLineConf	:FB_ReadXmlLine;
	FB_ReadXmlLineMsg	:FB_ReadXmlLine;

END_VAR
VAR_TEMP
	i					:INT;
END_VAR

VAR CONSTANT
	NO_OF_Torque		: INT :=50;
END_VAR
(*======================================================
   FB: fb_72x1_Achse (Achse ohne NC verfahren)
 ------------------------------------------------------
   Auth: 		Werner Friedl    						 
   Date: 		18.04.2018   						     
   Rev.: 		1.0	
   Desc:		siehe Aktion " Description "
 ========================================================*)
sub_connect();
sub_Visu();
IF 	NOT sHelp.b_init AND
	sConfig.Aktiv AND
	e_Position<> 0 AND
	Connect  THEN
	sHelp.b_init:=TRUE;
	sPos.r_18bit:=EXPT(2,18);		(*262144 für e_Velocity *)
	sPos.r_20bit:=EXPT(2,20);		(*1048576 für e_Position*)
	sPos.r_32bit:=EXPT(2,32);		(*4294967295 für Überlauf*)
	sConfig.UeberlaufControl_on:=sConfig.SW_Limit_on;
END_IF

IF	sConfig.Aktiv AND
	sConfig.Skalierfaktor <> 0 AND
	sConfig.Getriebefaktor <>0  AND
	sHelp.b_init AND
	Connect THEN
	sub_Regler();
	sub_Pos();
	sub_rec_Torque();
END_IF

Btn_init();
sub_ctrl();
sub_sdo();
sub_fb();

(* Toplevel *)
IF 	fb_state_entry.i16_next_step > INIT AND fb_state_entry.i16_next_step < FEHLER THEN
	IF 	sFb.ton_uez.Q AND NOT sCtrl.in.Fault THEN
		sSm.sm_timeout:=TRUE;
		fb_state_entry.i16_next_step := FEHLER;

	ELSIF
		sCtrl.in.Warning AND NotausOK THEN
		sSm.sm_Error_Warnung:=TRUE;
		fb_state_entry.i16_next_step := FEHLER;

	ELSIF
		fb_state_entry.i16_next_step >= BEREIT AND
		sCtrl.in.Fault THEN
		sSm.sm_Error_Klemme:=TRUE;
		fb_state_entry.i16_next_step := FEHLER;

	ELSIF
		fb_state_entry.i16_next_step >= BEREIT AND
		NOT Connect THEN
		sSm.sm_connect:=TRUE;
		fb_state_entry.i16_next_step := FEHLER;

	ELSIF
		sConfig.ModeOfOperation = CSV AND
		sFb.ton_uez_velo.Q THEN
		sSm.sm_Check_Velo:=TRUE;
	(*	stop:=TRUE;*)

(*	ELSIF fb_state_entry.i16_next_step >= BEREIT AND  sConfig.UeberlaufControl_on AND
		sPos.i32_count_ueberlauf <> 0 THEN
		sSm.sm_Ueberlauf:=TRUE;
		fb_state_entry.i16_next_step := FEHLER;*)
	ELSIF fb_state_entry.i16_next_step >= BEREIT AND  sConfig.Torque_Limit >0 AND
		sConfig.Torque_Limit > e_Torque THEN
		sSm.sm_Torque_zu_gross:=TRUE;
		fb_state_entry.i16_next_step := FEHLER;

	ELSIF sConfig.ModeOfOperation = CSP AND
		sPos.lr_MaxDiff > sConfig.max_PosDiff AND
		sConfig.PosDiffControl_on THEN
		sSm.sm_PosDiff:=TRUE;
		stop:=TRUE;
	END_IF
END_IF

(* ==================================Schrittkette================================ *)
fb_state_entry(	i16_pos:= 1);

CASE fb_state_entry.i16_step OF
(*=======================================================*)
INIT_OBJ:
	fb_state_entry.i16_next_step := INIT;

(*==========================================================================================================*)
INIT:
	IF	 fb_state_entry.E THEN

		sFb.ton_uez.IN := FALSE;
		sFb.ton_quitt.IN := FALSE;
		Stop:=FALSE;
		Reset:=FALSE;
		Busy:=FALSE;
		Error_:=FALSE;
		Done:=FALSE;
		Ready:=FALSE;
		on:=FALSE;

		sCtrl.out:=sCtrlEmpty.out;

	END_IF

		IF	sConfig.aktiv THEN
			fb_state_entry.i16_next_step := 20;
		ELSE
			fb_state_entry.i16_next_step := INAKTIV;
		END_IF

20:(*Switched_on*)

	IF	fb_state_entry.E THEN
		sCtrl.out.Fault_reset:=TRUE;
		sFb.ton_uez.IN:=TRUE;
	END_IF

	(*-----------------------Weiterschaltbedingungen----------------------------*)

	IF	NOT sCtrl.in.Fault THEN
		fb_state_entry.i16_next_step := BEREIT;
		sCtrl.out.Fault_reset:=FALSE;
	ELSE
		IF	sFb.ton_uez.Q THEN
			fb_state_entry.i16_next_step := FEHLER;
		END_IF
	END_IF

(*==========================================================================================================*)
BEREIT:
	IF	fb_state_entry.E THEN
		sFb.ton_uez.IN:=FALSE;
		Ready:=TRUE;
	END_IF

	IF	(sFb.r_trig_MotorOn.Q OR MotorOn)AND
		NOT on THEN
		IF 	NotausOK THEN
			MotorOn:=FALSE;
			sCtrl.out.Target_Position:=sCtrl.in.Position;
			fb_state_entry.i16_next_step := 110;
		ELSE
			sSm.sm_NotausNok:=TRUE;
			fb_state_entry.i16_next_step := FEHLER;
		END_IF
	END_IF

	CASE	sConfig.ModeOfOperation OF

	CSV:
			;
	CSP:
		(*Positionsübergabe*)

		IF 	on AND
			(*Positive Richtung*)
			 ((sVisuAxis.BtnJogP.Pressed AND sVisuAxis.b_kont) OR MoveP) THEN
			IF	sConfig.SW_Limit_on THEN
				IF	sCtrl.in.Position < sConfig.SW_Limit_max THEN
					sCtrl.out.Target_Position:=sConfig.SW_Limit_max;
				END_IF
			ELSE
				sCtrl.out.Target_Position:=sCtrl.in.Position+10000;
			END_IF
			Busy:=TRUE;
			Done:=FALSE;
		END_IF

		IF 	on AND
			(*Negative Richtung*)
			((sVisuAxis.BtnJogM.Pressed AND sVisuAxis.b_kont) OR MoveN) THEN
			IF	sConfig.SW_Limit_on THEN
				IF	sCtrl.in.Position > sConfig.SW_Limit_min THEN
					sCtrl.out.Target_Position:=sConfig.SW_Limit_min;
				END_IF
			ELSE
				sCtrl.out.Target_Position:=sCtrl.in.Position-10000;
			END_IF
			Busy:=TRUE;
			Done:=FALSE;
		END_IF

		(*Jog beenden*)
		IF	sFb.r_trig_jogP.Q OR sFb.r_trig_jogM.Q OR
			sFb.r_trig_MoveP.Q OR sFb.r_trig_MoveM.Q OR
			sFb.r_trig_stop.Q OR reset OR
			Stop  THEN
			Busy:=FALSE;
			Done:=TRUE;
			MoveP:=FALSE;
			MoveN:=FALSE;
			sCtrl.out.Target_Position:=sCtrl.in.Position;
		END_IF


		(*Positionieren mit Positionsvorgabe Absolut*)
		IF	on  AND
			(sFb.r_trig_MoveAbs.Q OR MoveAbs)THEN
			IF	sConfig.SW_Limit_on THEN
				IF	Vorgabe_Pos_Abs > sConfig.SW_Limit_max THEN
					sCtrl.out.Target_Position:=sConfig.SW_Limit_max;
					sSm.sm_SW_Limit:=TRUE;
				ELSIF	Vorgabe_Pos_Abs < sConfig.SW_Limit_min THEN
					sCtrl.out.Target_Position:=sConfig.SW_Limit_min;
					sSm.sm_SW_Limit:=TRUE;
				ELSE
					sCtrl.out.Target_Position:=Vorgabe_Pos_Abs;
					sSm.sm_SW_Limit:=FALSE;
				END_IF
			ELSE
				sCtrl.out.Target_Position:=Vorgabe_Pos_Abs;
			END_IF
			Busy:=TRUE;
			Done:=FALSE;
			bMove:=TRUE;
		END_IF

		(*Positionieren mit Positionsvorgabe Relativ*)
		IF	on  AND
			MoveRel THEN
			IF	sConfig.SW_Limit_on THEN
				IF	Vorgabe_Pos_Rel+sCtrl.out.Target_Position > sConfig.SW_Limit_max THEN
					sCtrl.out.Target_Position:=sConfig.SW_Limit_max;
					sSm.sm_SW_Limit:=TRUE;
				ELSIF	Vorgabe_Pos_Rel+sCtrl.out.Target_Position < sConfig.SW_Limit_min THEN
					sCtrl.out.Target_Position:=sConfig.SW_Limit_min;
					sSm.sm_SW_Limit:=TRUE;
				ELSE
					sCtrl.out.Target_Position:=sCtrl.out.Target_Position+Vorgabe_Pos_Rel;
					sSm.sm_SW_Limit:=FALSE;
				END_IF
			ELSE
				sCtrl.out.Target_Position:=sCtrl.out.Target_Position+Vorgabe_Pos_Rel;
			END_IF
			Busy:=TRUE;
			Done:=FALSE;
			bMove:=TRUE;
		END_IF
		IF	NOT on  AND
			(MoveAbs OR MoveRel)THEN
			fb_state_entry.i16_next_step := FEHLER;
		END_IF
	END_CASE

	(*Regler abschalten*)
	IF	(sFb.r_trig_reset.Q OR MotorOff OR NOT NotausOK )AND
		on	THEN
		sSm.sm_Move:=bMove;
		fb_state_entry.i16_next_step := 210;
	END_IF

	sFb.ton_Busy(IN:=Busy , PT:= t#50ms, Q=> , ET=> );
	IF	sFb.ton_Busy.Q AND On_Position AND
		fb_state_entry.i16_next_step = fb_state_entry.i16_step THEN
		Busy:=FALSE;
		Done:=TRUE;
		bMove:=FALSE;
		IF	sSm.sm_SW_Limit THEN
			fb_state_entry.i16_next_step := FEHLER;
		END_IF
	END_IF

	MotorOff:=FALSE;
	Stop:=FALSE;
	MoveAbs:=FALSE;
	MoveRel:=FALSE;

	IF	fb_state_entry.X THEN
		sFb.ton_uez.IN:=TRUE;
		Busy:=TRUE;
		Error_:=FALSE;
		Done:=FALSE;
		bMove:=FALSE;
	END_IF

(*==========================================================================================================*)
110:(*Ready_to_switch_on*)

	IF	fb_state_entry.E THEN
		sCtrl.out.Enable_voltage:=TRUE;
		sCtrl.out.Shutdown:=TRUE;
		sSm:=sSmEmpty;
	END_IF

	(*-----------------------Weiterschaltbedingungen----------------------------*)
	IF	sCtrl.in.Ready_to_switch_on THEN
		sCtrl.out.Switch_on:=TRUE;
		fb_state_entry.i16_next_step := 120;
	END_IF

(*=======================================================*)
120:(*Switched_on*)

	IF	fb_state_entry.E THEN
		sCtrl.out.Switch_on:=TRUE;
	END_IF

	(*-----------------------Weiterschaltbedingungen----------------------------*)

	IF	sCtrl.in.Switched_on THEN
		fb_state_entry.i16_next_step := 130;
	END_IF

130:(*Operation_enabled*)

	IF	fb_state_entry.E THEN
		sCtrl.out.Enable_operation:=TRUE;
	END_IF

	(*-----------------------Weiterschaltbedingungen----------------------------*)

	IF	sCtrl.in.Operation_enabled THEN
		fb_state_entry.i16_next_step := BEREIT;
		Busy:=FALSE;
		Error_:=FALSE;
		on:=TRUE;
	END_IF

(*==========================================================================================================*)
210:(*Switch_off*)

	IF	fb_state_entry.E THEN
		sCtrl.out.Target_Position:=sCtrl.in.Position;
		sCtrl.out.Enable_operation:=FALSE;
		sCtrl.out.Switch_on:=FALSE;
		on:=FALSE;
		MoveP:=FALSE;
		MoveN:=FALSE;
		Reset:=FALSE;
	END_IF

	(*-----------------------Weiterschaltbedingungen----------------------------*)

	IF	NOT sCtrl.in.Operation_enabled THEN
			fb_state_entry.i16_next_step := 220;
	END_IF

(*=======================================================*)
220:(*Shutdown*)

	IF	fb_state_entry.E THEN
		sCtrl.out.Shutdown:=FALSE;
	END_IF

	(*-----------------------Weiterschaltbedingungen----------------------------*)

	IF	NOT sCtrl.in.Ready_to_switch_on THEN
		fb_state_entry.i16_next_step := 230;
	END_IF

230:(*disabled_voltage*)

	IF	fb_state_entry.E THEN
			sCtrl.out.Enable_voltage:=FALSE;
	END_IF

	(*-----------------------Weiterschaltbedingungen----------------------------*)

	IF	sCtrl.in.Switch_on_disabled THEN
		sCtrl.out.Target_Position:=sCtrl.in.Position;
		fb_state_entry.i16_next_step := 240;
		Busy:=FALSE;
		Error_:=FALSE;
	END_IF

240:(**)
	IF	sSm.sm_PosDiff OR
		sSm.sm_Check_Velo OR
		sSm.sm_Move THEN
		fb_state_entry.i16_next_step := FEHLER;
	ELSE
		fb_state_entry.i16_next_step := BEREIT;
		sSm:=sSmEmpty;
	END_IF

(*==========================================================================================================*)
FEHLER: (*Fehler*)
	IF	fb_state_entry.E THEN
		Busy:=FALSE;
		Error_:=TRUE;
		Ready:=FALSE;
		on:=FALSE;
		MoveP:=FALSE;
		MoveN:=FALSE;
		sCtrl.out:=sCtrlEmpty.out;

		IF	sSm.sm_timeout THEN
			FB_ReadXmlLineMsg.ID:='sm_timeout';
			Error.No:=1;
		ELSIF	sSm.sm_Error_Klemme THEN
			FB_ReadXmlLineMsg.ID:='sm_Error_Klemme';
			Error.No:=2;
		ELSIF	sSm.sm_Error_Warnung THEN
			FB_ReadXmlLineMsg.ID:='sm_Error_Warnung';
			Error.No:=3;
		ELSIF	sSm.sm_Check_Velo THEN
			FB_ReadXmlLineMsg.ID:='sm_Check_Velo';
			Error.No:=4;
		ELSIF	sSm.sm_SW_Limit THEN
			FB_ReadXmlLineMsg.ID:='sm_SW_Limit';
			Error.No:=5;
		ELSIF		sSm.sm_PosDiff THEN
			FB_ReadXmlLineMsg.ID:='sm_PosDiff';
			Error.No:=6;
		ELSIF		sSm.sm_fehler_daten_schreiben THEN
			FB_ReadXmlLineMsg.ID:='sm_fehler_daten_schreiben';
			Error.No:=7;
		ELSIF		sSm.sm_connect THEN
			FB_ReadXmlLineMsg.ID:='sm_connect';
			Error.No:=8;
		ELSIF		sSm.sm_Ueberlauf THEN
			FB_ReadXmlLineMsg.ID:='sm_Ueberlauf';
			Error.No:=9;
		ELSIF			sSm.sm_Torque_zu_gross THEN
			FB_ReadXmlLineMsg.ID:='sm_Torque_zu_gross';
			Error.No:=10;
		ELSIF
			sSm.sm_NotausNok	THEN
			FB_ReadXmlLineMsg.ID:='sm_NotausNok';
			Error.No:=11;
		ELSIF
			sSm.sm_Move	THEN
			FB_ReadXmlLineMsg.ID:='sm_Move';
			Error.No:=12;
		END_IF

		Error.DateTime:=gVarDTSystemtime;

	END_IF

	sVisu.ProcessTime:=ProcessTime;

	IF	sFb.r_trig_quitt.Q THEN
			fb_state_entry.i16_next_step := INIT;
	END_IF

	IF sFb.ton_quitt.Q THEN
		sFb.ton_quitt(IN := FALSE);
	END_IF

INAKTIV:

	Busy:=FALSE;
	Ready := TRUE;
	Done := TRUE;

	IF	sConfig.aktiv THEN
		fb_state_entry.i16_next_step := FEHLER;
	END_IF

END_CASE

fb_state_entry(i16_pos:= 2);


(*------------------------------------------------------------------
	Error-Handling
  ------------------------------------------------------------------*)
IF	sVisuAxis.BtnReset.Pressed OR Reset THEN
	sSm:=sSmEmpty;
END_IF
IF	(MEMCMP(ADR(sSmEmpty), ADR(sSm), SIZEOF(sSmEmpty)) = 0 ) THEN
	Error.No:=0;
	Error.Text:='';
	TempErrorText:='';
END_IF
IF Error.Text<>''	AND ST_Lng.b_EndChangeLng THEN
	(*Error.DateTime:=;*)
	Error.Typ:=0;
	ErrorHandler.AddError(ErrorToAdd:=Error,
						sVisu:=Visu.ErrorHandler);
END_IF

IF	TempErrorText <>'' AND
	FIND(TempErrorText,'#')=0 AND
	LEN(TempErrorText)>40 THEN
	TempErrorText:=CONCAT(TempErrorText, '##');
END_IF

	LaufschriftObj(
	N:= 40,
	StepWidth:=1,
	PT:= t#100ms ,
	Text:= TempErrorText,
	Display=>sVisu.ErrorString );

	LaufschriftErrh(
	N:= 100,
	StepWidth:=1,
	PT:= t#100ms ,
	Text:= TempErrorText,
	Display=>Error.Text );

FB_ReadXmlLineConf(
	Prefix:= 'CONFIG',
	ID:= sConfig.InstName,
	File:= 'CONFIG.xml',
	Text=>  );

FB_ReadXmlLineMsg(
	Prefix:= 'MSG',
	ID:= ,
	File:= 'MSG.xml',
	Text=>);

IF	Error_ THEN
	TempErrorText:=CONCAT(sConfig.InstName,': ');
(*	TempErrorText:=CONCAT(TempErrorText,sConfig.Description);*)
	TempErrorText:=CONCAT(TempErrorText,FB_ReadXmlLineConf.Text);
	TempErrorText:=CONCAT(TempErrorText,' -> ');
	TempErrorText:=CONCAT(TempErrorText,FB_ReadXmlLineMsg.Text);
END_IF
END_FUNCTION_BLOCK
ACTION Btn_init:
(*Einheiten			===============================================================================*)
IF 	sConfig.Modulo THEN
	sVisuAxis.Einheit_pos:='°';
	sVisuAxis.Einheit_velo:='rpm ';
ELSE
	sVisuAxis.Einheit_pos:='mm';
	sVisuAxis.Einheit_velo:='mm/min';
END_IF
(*===================================================================================================*)

sVisuAxis.BtnReset.Text := 'Reset / Off';
sVisuAxis.BtnReset.Enable :=  ModeSelect.Mode <=MODE_MANUAL;
sVisuAxis.BtnReset.Visible := TRUE;
IF	sVisuAxis.BtnReset.Enable THEN
	sVisuAxis.BtnReset.TextColor := Color.black;
ELSE
	sVisuAxis.BtnReset.TextColor := Color.grey;
END_IF
IF	sVisuAxis.BtnReset.Pressed THEN
	sVisuAxis.BtnReset.BackgroundColor:=Color.darkgrey;
ELSE
	sVisuAxis.BtnReset.BackgroundColor:=Color.lightgrey;
END_IF
(*-------------------------------------------------------*)
sVisuAxis.BtnStop.Text := 'Stop';
sVisuAxis.BtnStop.Enable := On AND NOT Error_ AND NOT On_Position AND ModeSelect.Mode <=MODE_MANUAL ;
sVisuAxis.BtnStop.Visible := On AND NOT Error_ AND NOT On_Position AND ModeSelect.Mode <=MODE_MANUAL AND NOT sVisuAxis.BtnJogP.Pressed AND NOT sVisuAxis.BtnJogM.Pressed;
IF	sVisuAxis.BtnStop.Enable THEN
	sVisuAxis.BtnStop.TextColor := Color.black;
ELSE
	sVisuAxis.BtnStop.TextColor := Color.grey;
END_IF
IF	sVisuAxis.BtnStop.Pressed THEN
	sVisuAxis.BtnStop.BackgroundColor:=Color.darkgrey;
ELSE
	sVisuAxis.BtnStop.BackgroundColor:=Color.lightgrey;
END_IF
(*-------------------------------------------------------*)
sVisuAxis.BtnJogP.Text := '+';
sVisuAxis.BtnJogP.Enable := On AND (On_Position OR sVisuAxis.BtnJogP.Pressed) AND NOT Error_ AND ModeSelect.Mode <=MODE_MANUAL ;
IF	sVisuAxis.BtnJogP.Enable THEN
	sVisuAxis.BtnJogP.TextColor := Color.black;
ELSE
	sVisuAxis.BtnJogP.TextColor := Color.grey;
END_IF
sVisuAxis.BtnJogP.Visible := sConfig.ModeOfOperation=CSP;
IF	sVisuAxis.BtnJogP.Pressed THEN
	sVisuAxis.BtnJogP.BackgroundColor:=Color.yellow;
ELSE
	sVisuAxis.BtnJogP.BackgroundColor:=Color.lightgrey;
END_IF
(*-------------------------------------------------------*)
sVisuAxis.BtnJogM.Text := '-';
sVisuAxis.BtnJogM.Enable := On AND (On_Position OR sVisuAxis.BtnJogM.Pressed) AND NOT Error_ AND ModeSelect.Mode <=MODE_MANUAL ;
IF	sVisuAxis.BtnJogM.Enable THEN
	sVisuAxis.BtnJogM.TextColor := Color.black;
ELSE
	sVisuAxis.BtnJogM.TextColor := Color.grey;
END_IF
sVisuAxis.BtnJogM.Visible := sConfig.ModeOfOperation=CSP;
IF	sVisuAxis.BtnJogM.Pressed THEN
	sVisuAxis.BtnJogM.BackgroundColor:=Color.yellow;
ELSE
	sVisuAxis.BtnJogM.BackgroundColor:=Color.lightgrey;
END_IF
(*-------------------------------------------------------*)
sVisuAxis.BtnMotorOn.Text := 'Motor On';
sVisuAxis.BtnMotorOn.Enable := NOT On AND NOT Error_ AND ModeSelect.Mode <=MODE_MANUAL ;
IF	sVisuAxis.BtnMotorOn.Enable THEN
	sVisuAxis.BtnMotorOn.TextColor := Color.black;
ELSE
	sVisuAxis.BtnMotorOn.TextColor := Color.grey;
END_IF
sVisuAxis.BtnMotorOn.Visible := sConfig.ModeOfOperation=CSP;
IF	sVisuAxis.BtnMotorOn.Pressed THEN
	sVisuAxis.BtnMotorOn.BackgroundColor:=Color.darkgrey;
ELSE
	sVisuAxis.BtnMotorOn.BackgroundColor:=Color.lightgrey;
END_IF

(*-------------------------------------------------------*)
sVisuAxis.BtnMoveAbs.Text := 'Move Absolut';
sVisuAxis.BtnMoveAbs.Enable :=On AND On_Position AND NOT Error_ AND Vorgabe_Pos_Abs<>sCtrl.out.Target_Position  AND ModeSelect.Mode <=MODE_MANUAL ;
IF	sVisuAxis.BtnMoveAbs.Enable THEN
	sVisuAxis.BtnMoveAbs.TextColor := Color.black;
ELSE
	sVisuAxis.BtnMoveAbs.TextColor := Color.grey;
END_IF
sVisuAxis.BtnMoveAbs.Visible := sConfig.ModeOfOperation=CSP;
IF	sVisuAxis.BtnMoveAbs.Pressed THEN
	sVisuAxis.BtnMoveAbs.BackgroundColor:=Color.yellow;
ELSE
	sVisuAxis.BtnMoveAbs.BackgroundColor:=Color.lightgrey;
END_IF

(*-------------------------------------------------------*)
sVisuAxis.BtnTeach.Text := 'Teach';
sVisuAxis.BtnTeach.Enable :=On AND NOT Error_ AND On_Position  AND ModeSelect.Mode <=MODE_MANUAL ;
IF	sVisuAxis.BtnTeach.Enable THEN
	sVisuAxis.BtnTeach.TextColor := Color.black;
ELSE
	sVisuAxis.BtnTeach.TextColor := Color.grey;
END_IF
sVisuAxis.BtnTeach.Visible := sConfig.ModeOfOperation=CSP;
IF	sVisuAxis.BtnTeach.Pressed THEN
	sVisuAxis.BtnTeach.BackgroundColor:=Color.grey;
ELSE
	sVisuAxis.BtnTeach.BackgroundColor:=Color.lightgrey;
END_IF
END_ACTION
ACTION Description:
;(*======================================================
   FB: fb_72x1_Achse (Achse ohne NC verfahren)
 ------------------------------------------------------
   Auth: 		Werner Friedl    						 
   Date: 		18.04.2018   						     
   Rev.: 		1.0	
   Desc:		Mit diesem FB  können Antriebe ohne NC mit der PLC verfahren werden.
			- Die Struktur "sConfig" beinhaltet alle Variablen zur Motorkonfiguration.
			- über die VAR_INPUT	kann die Achse positioniert werden.
			  und über VAR_OUTPUT kann der Zustand abgefragt werden.
			  Beschreibung (siehe Variablendeklaration)	

			- Motor Bereit zum Einschalten: Ready
	
			- Motor einschalten:		MotorOn:=TRUE;
			- Motor ausschalten:  	MotorOff:=TRUE;

			- Abragen ob eingeschaltet:	On

--->			- Relative Bewegung (inkremental)
				Bewegung starten:	MoveRel:=TRUE; 
									Vorgabe_Pos_Rel:=100;
									Vorgabe_Velo:=1000;
				Bewegung gestartet:	Busy    
				Position erreicht :	Done

-->			- Absolute Bewegung
				Bewegung starten:	MoveAbs:=TRUE; 
									Vorgabe_Pos_Abs:=100;
									Vorgabe_Velo:=1000;
				Bewegung gestartet:	Busy    
				Position erreicht :	Done

-->			- Motor bewegen ohne Positionierung
			  (Softwarelimit abschalten sonst fährt die Achse nur bis zum Limit): 
									MoveP:=TRUE;	(positiv)
									MoveN:=TRUE	(negativ)
									Vorgabe_Velo:=1000;

				Bewegung gestartet:	Busy

	- Die Zählrichtunug des Messsystem wird im tsm eingestellt (Coe-Online 8000.01 
	- Die Globale CONSTANTE 	NO_OF_POS_AXIS  beschreibt die Anzahl der Positinen in der Positionsliste.
    	- in den TD kann eine Positionsliste angelegt werden. z.B.	
		TD.Posxxxxx	 			: ARRAY [1..NO_OF_POS_AXIS] OF st_Pos;	
	- in den MP muss ein PosOffset und ein Override angelegt werden.
		MP.xxxx.PosOffset_xxxx	 		: st_Pos;
		MP.xxxx.Override_xxxx			: DINT :=10;
	- für diesen FB gibt es ein Visuobjekt: 	ZLIB_7211_ACHSE
	- alle Strukturen im Ordner EL72x1 müssen vorhanden sein



Beispiel Initialisierung:

(*Init ST08_180_M1 Abstapeln*)
ST08_180_M1.sConfig.Description		:='Abstapeln';
ST08_180_M1.sConfig.InstName			:='ST08_180_M1';
ST08_180_M1.sConfig.Aktiv				:=TRUE;
ST08_180_M1.sConfig.Skalierfaktor		:=0.00034332275390625	;	(*360 / 1048576*)
ST08_180_M1.sConfig.Getriebefaktor		:=10;
ST08_180_M1.sConfig.Modulo			:=FALSE;
ST08_180_M1.sConfig.Pos_Faktor		:=5;				(*Weg bei einer Umdrehung in mm (nach Getriebe)*)
ST08_180_M1.sConfig.maxRpm			:=5338;
ST08_180_M1.sConfig.ModeOfOperation	:=CSP;			(*CSP,CSV,CST,CSTCA muss an der KLemme (Coe-Online 7010.03) eingestellt werden*)
(*nur für Coe-Online 7010.03 (CSP) position mode*)
ST08_180_M1.sConfig.RampTime		:=t#500ms;		(*Bauselle*)(*Beschleunigung und Bremsrampe*)
ST08_180_M1.sConfig.PosDiffControl_on	:=FALSE;		(*Baustelle*)
ST08_180_M1.sConfig.max_PosDiff		:=720;			(*Baustelle*)
ST08_180_M1.sConfig.SW_Limit_on		:=FALSE;
ST08_180_M1.sConfig.SW_Limit_min		:=-1000;
ST08_180_M1.sConfig.SW_Limit_max	:=1000;
ST08_180_M1.sConfig.lr_kp 				:= 800;
ST08_180_M1.sConfig.lr_ki 				:= 100.0;
ST08_180_M1.sConfig.lr_kd 				:= 50;

Beispiel Aufruf::

(*Call ST08_180_M1 Abstapeln*)
ST08_180_M1			(	sVisu:=	Visu.ST08_180_M1,
						Override:=	 MP.ST08.Override_Abstapeln,
						Offset:=		MP.ST08.PosOffsetAbstapeln.Pos,	(* in mm oder Grad am Abtrieb*)
						Reset:=		Visu.ModeSelect.BtnReset.Pressed );
IF	ST08_180_M1.sVisuAxis.BtnTeach.Pressed THEN
	TD.PosAbstapeln[ST08_180_M1.sVisuAxis.PosNr].Pos:= ST08_180_M1.sctrl.in.Position;
END_IF


 ===============================================================================================================================*)
END_ACTION
ACTION sub_connect:
IF	e_Toggle <> sHelp.b_ToggleHelp OR	(*die alten EL7211 haben kein e_Toggle, desshalb gibt es auch den e_State*)
	e_State = 8 THEN
	Connect:=TRUE;
	sHelp.b_ToggleHelp:=e_Toggle;
ELSE
	Connect:=FALSE;
END_IF
e_State:=e_State;(*
0x___1 = Slave in 'INIT' state
0x___2 = Slave in 'PREOP' state
0x___3 = Slave in 'BOOT' state
0x___4 = Slave in 'SAFEOP' state
0x___8 = Slave in 'OP' state
0x001_ = Slave signals error
0x002_ = Invalid vendorId, productCode... read
0x004_ = Initialization error occurred
0x008_ = Slave disabled
0x010_ = Slave not present
0x020_ = Slave signals link error
0x040_ = Slave signals missing link
0x080_ = Slave signals unexpected link
0x100_ = Communication port A
0x200_ = Communication port B
0x400_ = Communication port C
0x800_ = Communication port D*)
END_ACTION
ACTION sub_ctrl:
(*================================================================================================*)
(*Statusword*)
(*Bit  0*) sCtrl.in.Ready_to_switch_on:=		e_Statusword.0;
(*Bit 1 *) sCtrl.in.Switched_on:=			e_Statusword.1;
(*Bit 2 *) sCtrl.in.Operation_enabled	:=	e_Statusword.2;
(*Bit 3 *) sCtrl.in.Fault:=					e_Statusword.3;
(*Bit 4 *) 								e_Statusword.4;
(*Bit 5 *) 								e_Statusword.5;
(*Bit 6 *) sCtrl.in.Switch_on_disabled:=		e_Statusword.6;
(*Bit 7 *) sCtrl.in.Warning:=				e_Statusword.7;
(*Bit 8 *) 								e_Statusword.8;
(*Bit 9 *) 								e_Statusword.9;
(*Bit 10*) sCtrl.in.TxPDOToggle:=			e_Statusword.10; (*An-/Abwahl über 0x8010:01[} 136]*)
(*Bit 11*) sCtrl.in.Internal_Limit_active:=		e_Statusword.11;
(*Bit 12*) sCtrl.in.Target_value_ignored:=	e_Statusword.12;
(*Bit 13*) 								e_Statusword.13;
(*Bit 14*) 								e_Statusword.14;
(*Bit 15*) 								e_Statusword.15;

(*Controlword*)
(*Bit 0 *) a_Controlword.0:= sCtrl.out.Switch_on;
(*Bit 1 *) a_Controlword.1:= sCtrl.out.Enable_voltage;
(*Bit 2 *) a_Controlword.2:= sCtrl.out.Shutdown;
(*Bit 3 *) a_Controlword.3:= sCtrl.out.Enable_operation;
(*Bit 4 *) a_Controlword.4;
(*Bit 5 *) a_Controlword.5;
(*Bit 6 *) a_Controlword.6;
(*Bit 7 *) a_Controlword.7:= sCtrl.out.Fault_reset;
(*Bit 8 *) a_Controlword.8;
(*Bit 9 *) a_Controlword.9;
(*Bit 10*) a_Controlword.10;
(*Bit 11*) a_Controlword.11;
(*Bit 12*) a_Controlword.12;
(*Bit 13*) a_Controlword.13;
(*Bit 14*) a_Controlword.14;
(*Bit 15*) a_Controlword.15;
END_ACTION
ACTION sub_fb:
(* Zeiten *)
sFb.ton_uez		(IN:= ,PT:= t#3000ms, Q=>, ET=> );

sFb.ton_uez_velo	(IN:= sVelo.dif >15 AND on, PT:= t#300ms, Q=> , ET=> );
sFb.r_trig_Auto(CLK:=ModeSelect.Mode>MODE_MANUAL);
sFb.r_trig_Hand(CLK:=ModeSelect.Mode=MODE_MANUAL);
IF	sFb.r_trig_Hand.Q THEN
	sVisuAxis.Control:=TRUE;
ELSIF
	sFb.r_trig_Auto.Q THEN
	sVisuAxis.Control:=FALSE;
END_IF

(* Flanken *)
sFb.r_trig_stop(CLK:= NOT sVisuAxis.BtnStop.Pressed );
sFb.r_trig_reset(CLK:=NOT sVisuAxis.BtnReset.Pressed );
sFb.r_trig_MotorOn(CLK:=NOT sVisuAxis.BtnMotorOn.Pressed);
sFb.r_trig_jogP(CLK:= NOT sVisuAxis.BtnJogP.Pressed);
sFb.r_trig_jogM(CLK:=NOT sVisuAxis.BtnJogM.Pressed);
sFb.r_trig_MoveP(CLK:= NOT MoveP);
sFb.r_trig_MoveM(CLK:=NOT MoveN);
sFb.r_trig_MoveAbs(CLK:= NOT sVisuAxis.BtnMoveAbs.Pressed);

(*
sFb.ton_quitt		(IN:= ,PT:= t#100ms, Q=> , ET=> );
sFb.r_trig_quitt(CLK:=
			NOT On AND (*FEHLER wird dadurch automatisch quittiert*)
			NOT Reset AND
			NOT sVisuAxis.BtnReset.Pressed );
*)


sFb.ton_quitt(
		IN:=	NOT On AND (*FEHLER wird dadurch automatisch quittiert*)
				NOT Reset AND
				NOT sVisuAxis.BtnReset.Pressed ,
		PT:= 	t#200ms);
sFb.r_trig_quitt(CLK:=sFb.ton_quitt.Q);
END_ACTION
ACTION sub_Pos:
sPos.ist:=sctrl.in.Position;
(*===============================================================================*)
IF	(*config.Modulo OR*)
	sConfig.Pos_Faktor=0 THEN
	sConfig.Pos_Faktor:=1;
END_IF

(*Encoderüberlauf===================================================================================*)
sPos.lr_delta_ueberlauf:=ABS(sPos.lr_akt_alt - e_Position);

IF	sPos.lr_akt_alt >	(sPos.r_32bit - sPos.lr_delta_ueberlauf) AND						(*Überlauf bei 4294967295*)
	e_Position < sPos.lr_delta_ueberlauf THEN
	sPos.i32_count_ueberlauf:=	sPos.i32_count_ueberlauf +1;
ELSIF sPos.lr_akt_alt < sPos.lr_delta_ueberlauf AND									(*Überlauf bei 4294967295*)
	e_Position >(sPos.r_32bit - sPos.lr_delta_ueberlauf) THEN
	sPos.i32_count_ueberlauf:=	sPos.i32_count_ueberlauf -1;
END_IF
sPos.lr_akt_alt:= e_Position;

sPos.lr_Uebrlauf_Dist:=sPos.r_32bit * sConfig.Skalierfaktor;							(*Pos in Grad am Motor*)
sPos.lr_Uebrlauf_Dist:=sPos.lr_Uebrlauf_Dist/ sConfig.Getriebefaktor;					(*Pos in Grad am Getriebe*)

IF	NOT sConfig.Modulo THEN
	sPos.lr_Uebrlauf_Dist:=sPos.lr_Uebrlauf_Dist * (sConfig.Pos_Faktor/360);			(* Position in mm bei Linearachse*)
END_IF
sPos.lr_Uebrlauf_DistOne:=sPos.lr_Uebrlauf_Dist;

(*Positon auf Null stellen wenn der Überlauf erreicht ist*)
IF	sPos.i32_count_ueberlauf < - sConfig.Getriebefaktor THEN
	sCtrl.out.Target_Position:=sCtrl.out.Target_Position + (sConfig.Getriebefaktor * sPos.lr_Uebrlauf_DistOne );
	sPos.i32_count_ueberlauf:=sPos.i32_count_ueberlauf + LREAL_TO_DINT(sConfig.Getriebefaktor);
ELSIF  sPos.i32_count_ueberlauf >  sConfig.Getriebefaktor THEN
	sCtrl.out.Target_Position:=sCtrl.out.Target_Position - (sConfig.Getriebefaktor * sPos.lr_Uebrlauf_DistOne );
	sPos.i32_count_ueberlauf:=sPos.i32_count_ueberlauf - LREAL_TO_DINT(sConfig.Getriebefaktor);
END_IF

sPos.lr_Uebrlauf_Dist:=sPos.lr_Uebrlauf_Dist *DINT_TO_LREAL(sPos.i32_count_ueberlauf);

(*Multiturn======================================================================================*)

sConfig.Skalierfaktor;
sCtrl.in.Position:=UDINT_TO_LREAL(e_Position )*sConfig.Skalierfaktor;	(*Pos in Grad am Motor*)
(*sPos.lr_Mod:=LMOD(sCtrl.in.Position ,config.Modulofaktor);		(*Moduloposition*)*)
sCtrl.in.Position:=sCtrl.in.Position/ sConfig.Getriebefaktor;					(*Pos in Grad am Getriebe*)
sPos.lr_Mod:=LMOD((sCtrl.in.Position-Offset) ,360);			(*Pos in Grad 0° - 360° *)

IF	NOT sConfig.Modulo THEN
	sCtrl.in.Position:=sCtrl.in.Position * (sConfig.Pos_Faktor/360);			(* Position in mm bei Linearachse*)

	sPos.lr_Target:=sCtrl.out.Target_Position / (sConfig.Pos_Faktor/360) ;	(*Pos in Grad am Getriebe° *)
	sPos.lr_Offset_Ink:=Offset / (sConfig.Pos_Faktor/360) ;		 (*OffsetPos in Grad am Getriebe° *)
ELSE
	sPos.lr_Target:=sCtrl.out.Target_Position;
END_IF

sCtrl.in.Position:=sPos.lr_Uebrlauf_Dist+sCtrl.in.Position-Offset;

sPos.lr_Target:=sPos.lr_Target * sConfig.Getriebefaktor;				(*Pos in Grad am Motor° *)
sPos.lr_Offset_Ink:=sPos.lr_Offset_Ink* sConfig.Getriebefaktor;			(*OffsetPos in Grad am Motor° *)
sPos.i32_Offset_Ink:=LREAL_TO_UDINT(sPos.lr_Offset_Ink / sConfig.Skalierfaktor);		(*OffsetPos in Inkrementen am Motor° *)
a_Target_Position:=LREAL_TO_UDINT(sPos.lr_Target / sConfig.Skalierfaktor);	(*Pos in Inkrementen am Motor° *)

a_Target_Position:=a_Target_Position-sPos.i32_Offset_Ink;
e_Position;


(*Singelturn===Baustelle========================================================================*)
sPos.lr_ModuloPosInc:=LMOD(e_Position ,sPos.r_20bit);			(*Moduloposition in Ikrementen*)

sPos.lr_ModuloHelp:=(e_Position - LREAL_TO_UDINT(sPos.lr_ModuloPosInc)) / LREAL_TO_UDINT(sPos.r_20bit) ;
sPos.lr_ModuloHelp2:=(e_Position - LREAL_TO_UDINT(sPos.lr_ModuloPosInc)) / LREAL_TO_UDINT(sPos.r_20bit) ;
sPos.i16_ModuloHelp:=GANZE_ZAHL(sPos.lr_ModuloHelp2 / sConfig.Getriebefaktor);
sPos.lr_ModuloCount:=sPos.lr_ModuloHelp2 - (sPos.i16_ModuloHelp * sConfig.Getriebefaktor);

sPos.lr_Pos:= (sPos.lr_ModuloCount * sPos.r_20bit)+sPos.lr_ModuloPosInc;
sPos.lr_Pos:=sPos.lr_Pos* sConfig.Skalierfaktor;				(*Pos in Grad am Motor*)
sPos.lr_Pos:=sPos.lr_Pos / sConfig.Getriebefaktor;				(*Pos in Grad am Getriebe*)
sPos.lr_Pos:=LMOD(sPos.lr_Pos ,360);							(*Pos in Grad 0° - 360° *)
sPos.lr_Pos:=sPos.lr_Pos * (sConfig.Pos_Faktor/360);			(* Position in mm bei Linearachse*)



(*Schleppfehler===================================================================================*)
sCtrl.in.Following_Error:=DINT_TO_LREAL(e_Following_Error)*sConfig.Skalierfaktor;

sFb.ton_aufPos(
		IN:= ABS(sCtrl.out.Target_Position - sCtrl.in.Position) <1,
		PT:=t#20ms,
		Q=>On_Position);
END_ACTION
ACTION sub_rec_Torque:
IF	ABS(e_Torque) > Torque[1] THEN
	i:=1;
	FOR i:=NO_OF_Torque TO 2 BY-1 DO
	   Torque[i] := Torque[i-1];
	END_FOR
	 Torque[1]:=ABS(e_Torque);
END_IF
END_ACTION
ACTION sub_Regler:
sPos.r_18bit;
sVelo.Faktor:=sPos.r_18bit / 60;
(*=============================================================================================================*)

sVelo.maxRpmNachGertiebe	:=sConfig.maxRpm/ sConfig.Getriebefaktor;		(*Maximale Drehzahl nach Getriebe*)
sVelo.maxLinear		:=sVelo.maxRpmNachGertiebe * sConfig.Pos_Faktor;		(*Maximale Geschwindigkeit in mm/min*)
IF	 sConfig.Modulo THEN
	sVelo.maxRpm:=sVelo.maxRpmNachGertiebe;	(*rpm*)
	sVelo.Vorgabe_Velo_rpm:=Vorgabe_Velo * LREAL_TO_INT(sConfig.Getriebefaktor);
ELSE
	sVelo.maxRpm:=sVelo.maxLinear;			(*mm/min*)
	sVelo.Vorgabe_Velo_rpm:=Vorgabe_Velo / sConfig.Pos_Faktor;
	sVelo.Vorgabe_Velo_rpm:=sVelo.Vorgabe_Velo_rpm * LREAL_TO_INT(sConfig.Getriebefaktor);
END_IF

IF	Vorgabe_Velo > sVelo.maxRpm THEN
	Vorgabe_Velo:= LREAL_TO_INT(sVelo.maxRpm);
END_IF

sRegler.lr_Override:=DINT_TO_LREAL(override)/100;
sVelo.ist:=e_Velocity / sVelo.Faktor;				(*rpm am Motor*)
sVelo.ist:=sVelo.ist / sConfig.Getriebefaktor;		(*rpm nach Getriebe*)
sVelo.soll:=sVelo.sollRpm / sConfig.Getriebefaktor;	(*rpm nach Getriebe*)
IF	 NOT sConfig.Modulo THEN
	sVelo.ist:=sVelo.ist * sConfig.Pos_Faktor;		(*Geschwindigkeit in mm/min*)
	sVelo.soll:=sVelo.soll * sConfig.Pos_Faktor;	(*Geschwindigkeit in mm/min*)
END_IF

sVelo.dif:=									(*rpm oder mm*)
	ABS(sVelo.soll-sVelo.ist);

IF 	NOT sHelp.b_init2 AND sVelo.maxRpm<>0 THEN
	Vorgabe_Velo:=LREAL_TO_DINT(sVelo.maxRpm);
	sHelp.b_init2:=TRUE;
END_IF
sCtrl.in.Velocity:=sVelo.ist;
(*=============================================================================================================*)
CASE	sConfig.ModeOfOperation OF

CSV:
	sVelo.sollRpm:=LREAL_TO_INT(sVelo.Vorgabe_Velo_rpm * sRegler.lr_Override);

CSP:

	sRegler.lr_delta :=
			sCtrl.out.Target_Position -
			sCtrl.in.Position; (* Grad *)
	sRegler.lr_delta :=	sRegler.lr_delta * sConfig.Getriebefaktor;
	IF	NOT sConfig.Modulo THEN
 		sRegler.lr_delta:=sRegler.lr_delta / (sConfig.Pos_Faktor/360);
	END_IF

	sRegler.lr_tmp := sRegler.lr_delta;
	IF (sRegler.lr_tmp > 10000) THEN
		sRegler.lr_tmp := 10000;
	END_IF
	IF (sRegler.lr_tmp < -10000) THEN
		sRegler.lr_tmp := -10000;
	END_IF

	sRegler.lr_current_p := 0.004  * sConfig.lr_kp * sRegler.lr_tmp ; (*  RPM *)
	sRegler.lr_current_i := sRegler.lr_current_i + 0.004  * sConfig.lr_ki * sRegler.lr_tmp ; (*  RPM *)
	sRegler.lr_current_d := 0.004  * sConfig.lr_kd * (sRegler.lr_tmp-sRegler.lr_delta_alt) ; (*  RPM *)

	IF (sRegler.lr_current_i > 1000) THEN
		sRegler.lr_current_i := 1000;
	END_IF
	IF (sRegler.lr_current_i < -1000) THEN
		sRegler.lr_current_i := -1000;
	END_IF
	(*----------------------------------------------------------*)
	sRegler.lr_delta_dif:=sRegler.lr_delta_alt - sRegler.lr_delta;
	sPos.lr_DiffPuls:=ABS(sRegler.lr_delta_dif) ;
	sPos.lr_DiffPuls:=sPos.lr_DiffPuls*sConfig.Skalierfaktor;
	sPos.lr_DiffVelo:=ABS(sVelo.sollRpm/60*360/1000*4);
	(*sPos.lr_DiffPuls:=sPos.lr_DiffPuls-sPos.lr_DiffVelo;*)

	IF	sPos.lr_MaxDiff < sPos.lr_DiffPuls THEN
		sPos.lr_MaxDiff := sPos.lr_DiffPuls;
	END_IF
	IF	sPos.lr_DiffPuls = 0 AND on THEN
		sPos.lr_MaxDiff := 0;
	END_IF
	(*----------------------------------------------------------*)

	IF	sRegler.lr_targetpos_alt<>sCtrl.out.Target_Position THEN
		sRegler.lr_delta_targetpos:=ABS(sRegler.lr_targetpos_alt - sCtrl.out.Target_Position);
		sRegler.lr_targetpos_alt:=sCtrl.out.Target_Position;
		sFb.ton_aufPos.IN:=FALSE;
	END_IF

	(*----------------------------------------------------------*)

	sRegler.lr_delta_alt :=sRegler.lr_tmp;

	sRegler.lr_current_v :=sRegler.lr_current_p +sRegler.lr_current_i +sRegler.lr_current_d;
	sVelo.Vorgabe_Velo_rpm;
	IF (sRegler.lr_current_v >sVelo.Vorgabe_Velo_rpm) THEN
		sRegler.lr_current_v := sVelo.Vorgabe_Velo_rpm;
	ELSIF (sRegler.lr_current_v < -sVelo.Vorgabe_Velo_rpm) THEN
		sRegler.lr_current_v := -sVelo.Vorgabe_Velo_rpm;
	END_IF

	sRegler.lr_current_v :=sRegler.lr_current_v ;

	IF	sRegler.lr_delta_targetpos >= 360 THEN
		IF	(ABS(sRegler.lr_delta) < 360) THEN
			sRegler.lr_current_v :=sRegler.lr_current_v * (ABS(sRegler.lr_delta) / 360);
		END_IF
	ELSE
		sRegler.lr_current_v := sRegler.lr_current_v * (ABS(sRegler.lr_delta) / 180);
	END_IF
	IF 	On_Position THEN
		sRegler.lr_delta_targetpos := 360;
	END_IF

	sVelo.sollRpm := LREAL_TO_DINT(sRegler.lr_current_v);

END_CASE


(*Beschränken auf Vorgabe*)

IF	sVelo.sollRpm > sVelo.Vorgabe_Velo_rpm THEN
	sVelo.sollRpm :=LREAL_TO_INT(sVelo.Vorgabe_Velo_rpm);
END_IF

IF	sVelo.sollRpm < sVelo.Vorgabe_Velo_rpm*(-1) THEN
	sVelo.sollRpm :=LREAL_TO_INT(sVelo.Vorgabe_Velo_rpm*(-1));
END_IF

sVelo.sollRpm:=sVelo.sollRpm * sRegler.lr_Override;

(*Ausgaber an Regler*)
IF 	on THEN
	a_Target_Velocity:=
		LREAL_TO_DINT(
		sVelo.sollRpm *
		 sVelo.Faktor) ;
ELSE
	a_Target_Velocity:=0;
END_IF
e_Velocity;
END_ACTION
ACTION sub_sdo:
(*=============================================================================================*)
sSdo.s_SlaveNetId:='172.18.137.69.4.1';
sSdo.ui16_SlaveAddr:=1012;
sSdo.i8_SubIndex:=0;
sSdo.w_Index:=16#8000;

(* Einen neuen EcCoeSdo-Parameter auf den Antrieb schreiben *)
sSdo.fb_ec_coe_sdo_write_ex(
	sNetId:= sSdo.s_SlaveNetId,
	nSlaveAddr:= sSdo.ui16_SlaveAddr,
	nSubIndex:= sSdo.i8_SubIndex,
	nIndex:= sSdo.w_Index,
	pSrcBuf:= ADR(sSdo.acObjectData),
	cbBufLen:= SIZEOF(sSdo.acObjectData),
	bExecute:= ,
	tTimeout:= t#10s,
	bCompleteAccess:= FALSE,
	bBusy=> ,
	bError=> ,
	nErrId=> );

(*=============================================================================================*)
(* Einen neuen EcCoeSdo-Parameter von dem Antrieb lesen *)
sSdo.fb_ec_coe_sdo_read_ex(
	sNetId:= sSdo.s_SlaveNetId,
	nSlaveAddr:= sSdo.ui16_SlaveAddr,
	nSubIndex:= sSdo.i8_SubIndex,
	nIndex:= sSdo.w_Index,
	pDstBuf:=  ADR(sSdo.acObjectData),
	cbBufLen:= SIZEOF(sSdo.acObjectData),
	bExecute:= ,
	tTimeout:= t#10s,
	bCompleteAccess:= FALSE,
	bBusy=> ,
	bError=> ,
	nErrId=> );
END_ACTION
ACTION sub_Visu:
sFb.r_trig_kont(CLK:= sVisuAxis.b_kont, Q=> );
sFb.r_trig_ink_10(CLK:= sVisuAxis.b_ink_10, Q=> );
sFb.r_trig_ink_100(CLK:= sVisuAxis.b_ink_100, Q=> );
sFb.r_trig_ink_1000(CLK:= sVisuAxis.b_ink_1000, Q=> );
sFb.r_trig_ink_var(CLK:= sVisuAxis.b_ink_var, Q=> );

IF	sFb.r_trig_kont.Q THEN
	sVisuAxis.b_ink_10:=FALSE;
	sVisuAxis.b_ink_100:=FALSE;
	sVisuAxis.b_ink_1000:=FALSE;
	sVisuAxis.b_ink_var:=FALSE;
ELSIF
	sFb.r_trig_ink_10.Q THEN
	sVisuAxis.b_kont:=FALSE;
	sVisuAxis.b_ink_100:=FALSE;
	sVisuAxis.b_ink_1000:=FALSE;
	sVisuAxis.b_ink_var:=FALSE;
ELSIF
	sFb.r_trig_ink_100.Q THEN
	sVisuAxis.b_kont:=FALSE;
	sVisuAxis.b_ink_10:=FALSE;
	sVisuAxis.b_ink_1000:=FALSE;
	sVisuAxis.b_ink_var:=FALSE;
ELSIF
	sFb.r_trig_ink_1000.Q THEN
	sVisuAxis.b_kont:=FALSE;
	sVisuAxis.b_ink_10:=FALSE;
	sVisuAxis.b_ink_100:=FALSE;
	sVisuAxis.b_ink_var:=FALSE;
ELSIF
	sFb.r_trig_ink_var.Q THEN
	sVisuAxis.b_kont:=FALSE;
	sVisuAxis.b_ink_10:=FALSE;
	sVisuAxis.b_ink_100:=FALSE;
	sVisuAxis.b_ink_1000:=FALSE;
ELSIF
	NOT sVisuAxis.b_kont AND
	NOT sVisuAxis.b_ink_10  AND
	NOT sVisuAxis.b_ink_100 AND
	NOT sVisuAxis.b_ink_1000 AND
	NOT sVisuAxis.b_ink_var THEN
	sVisuAxis.b_kont:=TRUE;
END_IF


IF	(sFb.r_trig_jogP.Q OR sFb.r_trig_jogM.Q) AND
	NOT sVisuAxis.b_kont THEN

	IF	sVisuAxis.b_ink_10  THEN
		Vorgabe_Pos_Rel:=0.01;
	ELSIF
		sVisuAxis.b_ink_100 THEN
		Vorgabe_Pos_Rel:=0.1;
	ELSIF
		sVisuAxis.b_ink_1000 THEN
		Vorgabe_Pos_Rel:=1;
	ELSIF
		sVisuAxis.b_ink_var THEN
		Vorgabe_Pos_Rel:=sVisuAxis.lr_ink_var;
	END_IF

	IF	sFb.r_trig_jogM.Q THEN
		Vorgabe_Pos_Rel:=Vorgabe_Pos_Rel * (-1);
	END_IF
	MoveRel:=TRUE;
END_IF

(*Positon aktivieren=======================================================*)
FOR i := -1 TO NO_OF_POS_AXIS  BY 1DO
	IF	sVisuAxis.b_Pos_nr[i] THEN
		sVisuAxis.PosNr:=i;
		Vorgabe_Pos_Abs:=sPosList[i].Pos;
	END_IF
END_FOR
sVisuAxis.b_Pos_nr:=sHelp.b_Pos_nr_Empty;


IF	sHelp.Pos <> sPosList[sVisuAxis.PosNr].Pos OR
	sHelp.PosNr <> sVisuAxis.PosNr OR
	 sVisuAxis.b_PosNr THEN
	Vorgabe_Pos_Abs:=sPosList[sVisuAxis.PosNr].Pos;
END_IF
sHelp.PosNr:=sVisuAxis.PosNr;
sHelp.Pos:=sPosList[sVisuAxis.PosNr].Pos;
END_ACTION

(* POU zLibrary/_HelpFunctions/FB_Laufschrift, ST *)
FUNCTION_BLOCK FB_Laufschrift
VAR_INPUT
	N 						:INT; (* Max output Stringlength *)
	StepWidth				:INT:=1;
	PT 						:TIME;
	Text 					:STRING; (* Original String *)
END_VAR
VAR_OUTPUT
	Display 					:STRING(255); (* Output String *)
END_VAR
VAR
	delay 					:TP;
	TempOutputString		:STRING(255);
	TempInputText			:STRING(255);
	step 					:INT;
END_VAR
(* generate next ticker when delay is low *)
IF 	N < LEN(text) THEN
	IF 	NOT delay.Q THEN
		(* increase step for next tick *)
		TempInputText:=text;
		step := step + StepWidth;

		IF step > LEN(TempInputText) THEN
			step := 1;
		END_IF

		(* extract dispay from text *)
		TempOutputString := MID(TempInputText, N, step);

		IF 	LEN(TempOutputString)<N THEN
			TempOutputString:=CONCAT(TempOutputString,TempInputText);
			TempOutputString:=LEFT(TempOutputString,N);
			Display:=TempOutputString;
		ELSE
			Display:=TempOutputString;
		END_IF
		(* set delay timer for next tick *)
		delay(IN := TRUE, PT := PT);
	ELSE
		(* execute delay timer *)
		delay(in := FALSE);
	END_IF
ELSE
	display := text;
END_IF
END_FUNCTION_BLOCK

(* POU zLibrary/ept/Achse/GANZE_ZAHL, ST *)
FUNCTION GANZE_ZAHL : INT
VAR_INPUT
	lr_Wert		:LREAL;
END_VAR
VAR
	st_Wert		:STRING;
	pos			:INT;
END_VAR
IF	lr_Wert >= 1 THEN

	st_Wert:=LREAL_TO_STRING(lr_Wert);
	pos:=FIND(st_Wert,'.');
	
	st_Wert:=LEFT(st_Wert,pos);
	
	GANZE_ZAHL:=STRING_TO_INT(st_Wert);
ELSE
	GANZE_ZAHL:=0;
END_IF
END_FUNCTION

(* POU zLibrary/AnaIn/FB_AnaInDint, ST *)
FUNCTION_BLOCK FB_AnaInDint
VAR_INPUT
	sInit					:sAnaInInit;	(* Initializingvalues to the Instance *)
END_VAR
VAR_OUTPUT
	State					:StateObject;	(* State of the object *)
	HomePosition			:BOOL;			(* object in home-position*)
	Value					:REAL;
END_VAR
VAR_IN_OUT
	sVisu					:sAnaInVisu;
END_VAR
VAR
	AnaInValue		AT %I* 	:DINT;			(* Ana in value *)

	Error					:ErrorStruct;
	TempErrorText			:STRING(255);
	InitState				:BOOL:=FALSE;	(* Internal State for initialising *)

	diffSource				:REAL;
	diffTarget				:REAL;

	FB_ReadXmlLineConf		:FB_ReadXmlLine;
	FB_ReadXmlLineMsg		:FB_ReadXmlLine;
END_VAR
Error.No:=0;
Error.Text:='';

(*------------------------------------------------------------------
	Initialization
  ------------------------------------------------------------------*)
IF  NOT InitState THEN
	InitState:=TRUE;

	(* Check instance name *)
	IF sInit.InstName=''THEN
		InitState:=FALSE;
		State:=STATE_ERROR;
		FB_ReadXmlLineMsg.ID:='InstNameNotDefined';

		TempErrorText:=sInit.BitInName;
		TempErrorText:=CONCAT(TempErrorText,' :');
		TempErrorText:=CONCAT(TempErrorText,sVisu.Description);
  		TempErrorText:=CONCAT(TempErrorText,' -> ');
		TempErrorText:=CONCAT(TempErrorText,FB_ReadXmlLineMsg.Text);
		Error.No:=4;
		(*Error.Text:='InstName not defined';*)
	(*CheckDescription*)
	ELSIF
		sInit.Description=''THEN
		InitState:=FALSE;
		State:=STATE_ERROR;
		FB_ReadXmlLineMsg.ID:='DescriptionNotDefined';

		TempErrorText:=sInit.BitInName;
		TempErrorText:=CONCAT(TempErrorText,' :');
		TempErrorText:=CONCAT(TempErrorText,sVisu.Description);
  		TempErrorText:=CONCAT(TempErrorText,' -> ');
		TempErrorText:=CONCAT(TempErrorText,FB_ReadXmlLineMsg.Text);
		Error.No:=4;
		(*Error.Text:='Description not defined';*)
	END_IF

	sVisu.InstName		:= sInit.InstName;
	sVisu.Description	:= sInit.Description;
	sVisu.ErrorString	:= Error.Text;
END_IF

(* Add InitState to Global-Init-State to collect all Objects *)
gInitCollect:=gInitCollect AND InitState;

IF 	InitState THEN
	diffSource := sinit.ScalingSensorValueMax - sinit.ScalingSensorValueMin;
  	diffTarget := sinit.ScalingOutputValueMax - sinit.ScalingOutputValueMin;
 	(*Value := (((AnaInValue-sinit.ScalingOutputValueMin)/diffSource)*diffTarget)+sinit.ScalingOutputValueMin;*)
 	Value :=  (AnaInValue- sinit.ScalingSensorValueMin) / (diffSource  / diffTarget) ;

	sVisu.AnaInValue:=Value;

END_IF
(* ------------------------------------------------------------------------------------------ *)
(* ---------------- LANGUAGE auslesen aus der XML Datei-------- *)
(* ------------------------------------------------------------------------------------------ *)
sVisu.BitInName:=sInit.BitInName;
sVisu.InstName:=sInit.InstName;
sVisu.ErrorPresent:=Error.Text<>'';

FB_ReadXmlLineConf(
	Prefix:= 'CONFIG',
	ID:= sInit.InstName,
	File:= 'CONFIG.xml',
	Text=> sVisu.Description  );


FB_ReadXmlLineMsg(
	Prefix:= 'MSG',
	ID:= ,
	File:= 'MSG.xml',
	Text=>);

IF 	State = STATE_ERROR THEN
	TempErrorText:=sInit.BitInName;
	TempErrorText:=CONCAT(TempErrorText,' :');
	TempErrorText:=CONCAT(TempErrorText,sVisu.Description);
	TempErrorText:=CONCAT(TempErrorText,' -> ');
	TempErrorText:=CONCAT(TempErrorText,FB_ReadXmlLineMsg.Text);
END_IF
END_FUNCTION_BLOCK

(* POU zLibrary/ept/Achse/fb_Auto_On_Off, ST *)
FUNCTION_BLOCK fb_Auto_On_Off
VAR_INPUT
	b_Stop				:BOOL;
END_VAR
VAR_IN_OUT
	Achse				:fb_72x1_Achse;
END_VAR
VAR
	fb_ton_wz			:TON;
	fb_ton_uez			:TON;

	fb_state_entry		:ST_StateEntry;
END_VAR
fb_ton_wz		(IN:= ,PT:= , Q=>  , ET=> );
fb_ton_uez		(IN:= ,PT:= t#2000ms, Q=>, ET=> );

(* ==================================Schrittkette================================ *)
fb_state_entry(	i16_pos:= 1);

CASE fb_state_entry.i16_step OF
(*=======================================================*)
INIT_OBJ:
	fb_state_entry.i16_next_step := INIT;

(*==========================================================================================================*)
INIT:
	fb_state_entry.i16_next_step := BEREIT;

(*==========================================================================================================*)
BEREIT:
	IF	fb_state_entry.E THEN
		;
	END_IF

	IF	ModeSelect.Mode=MODE_AUTO OR
		ModeSelect.Mode=MODE_AUTO_RUN OR
		ModeSelect.Mode=MODE_STEP_RUN THEN

		IF	NOT Achse.On AND
			NOT b_Stop AND
			NOT Achse.Error_ THEN
			Achse.MotorOn:=TRUE;
		END_IF

		fb_ton_uez.IN:=Achse.MotorOn;

		IF	b_Stop AND Achse.MotorOn THEN
			Achse.MotorOn:=FALSE;
			Achse.MotorOff:= TRUE;
		END_IF

	END_IF

(*==========================================================================================================*)
FEHLER: (*Fehler*)
	IF	fb_state_entry.E THEN
		;
	END_IF

END_CASE

fb_state_entry(i16_pos:= 2);
END_FUNCTION_BLOCK

(* POU zLibrary/DigIn/FB_DigIn, ST *)
FUNCTION_BLOCK FB_DigIn

VAR_OUTPUT
	State						: StateObject;	(* State of the object *)
	HomePosition				: BOOL;			(* object in home-position*)
	SignalIn						: BOOL;			(* Static signal of digital input *)
	SignalInDelayed				: BOOL;			(* Static signal of digital input but with on and of delay times *)
END_VAR
VAR_INPUT
	CheckSignalHigh			: BOOL;		 	(* Signal check  HIGH *)
	CheckSignalLow			: BOOL;		 	(* Signal check  LOW  *)

	Reset						: BOOL;			(* switch for resetting the control *)

	SFCCurrentStep				: STRING(40);	(* aktually step in the order of events *)
	SFCCurrentPOU				: STRING(40);	(* Name of the order of events*)

	sInit						: sDigInInit;		(* Initializingvalues to the Instance *)
END_VAR
VAR_IN_OUT
	sVisu						: sDigInVisu;
END_VAR
VAR
	BitInToCheck				AT %I* :BOOL;		(* Bit input signal to check *)

	ProcessTime					: DINT;					(* Counts the time in steps of 100ms since starting operation *)

	TimerTimeOut				: CheckProcTime;		(* Timer generates timeout signal *)
	Error						: ErrorStruct;
	ErrorElapsed				: BOOL;
	TempErrorText				: STRING(255);
	HomePositionInfo			: DINT;							(* missing to home posistion *)
	ResetIntern					: BOOL;							(* Internal reset signal *)


	BtnReset					: VisuButton;			(* Manage button *)

	StateOK_CycleFlag			: BOOL;

	FirstCheckCycle				:  R_TRIG;

	IputOnDelayTime				: TON;
	IputOffDelayTime			: TOF;

	(* --------------------------------------------------------------------------------- *)
	(*         Internal Variables	Visu				                                           *)
	(* --------------------------------------------------------------------------------- *)
	LaufschriftErrh				:FB_Laufschrift;
	LaufschriftObj				:FB_Laufschrift;

	FB_ReadXmlLineConf		:FB_ReadXmlLine;
	FB_ReadXmlLineMsg		:FB_ReadXmlLine;

END_VAR
Error.No:=0;
Error.Text:='';
TempErrorText:='';

(*------------------------------------------------------------------
	Initialization
  ------------------------------------------------------------------*)


(* Add InitState to Global-Init-State to collect all Objects *)
gInitCollect:=gInitCollect ;

IF gInitOk THEN

StateOK_CycleFlag := State=State_ok;


(*------------------------------------------------------------------
	Show and Read Buttons
  ------------------------------------------------------------------*)

BtnReset(	Button:=sVisu.BtnReset,
					Enable:=TRUE ,
					Visible:=ModeSelect.Mode=MODE_MANUAL,
					TextOn:='Reset',
					TextOff:='Reset',
					PressedExt:=FALSE ,
					StateOn:= FALSE ,
					);

	(*------------------------------------------------------------------
	Manual-Mode
  ------------------------------------------------------------------*)
	IF  ModeSelect.Mode=MODE_MANUAL THEN

		SFCCurrentStep:=sInit.InstName;
		SFCCurrentPOU:='MODE_MANUAL';
	END_IF (*ModeSelect.Mode=MODE_MANUAL*)


	(*reset timer in first cycle of checking*)
	FirstCheckCycle(CLK := CheckSignalHigh OR CheckSignalLow );

	IF 	FirstCheckCycle.Q THEN
		ProcessTime:=TimerTimeOut.PTime;
	END_IF

	(*------------------------------------------------------------------
	Mode higher manual mode (auto, tip or homeposrun)
  ------------------------------------------------------------------*)
	 	IF	( ModeSelect.Mode>MODE_MANUAL OR sInit.EnableInEveryMode) AND
			( CheckSignalHigh OR CheckSignalLow )	THEN

		(* Check input signal                                      *)
		(*=========================================================*)

		(* Check signal low and input is low*)
		IF 	NOT BitInToCheck AND
			CheckSignalLow AND
			NOT CheckSignalHigh THEN
			(* Check input low and it is low *)
			TimerTimeOut(Start := FALSE, MTime := (sInit.MaxTime));
			State:=State_OK;

		(* Check input low and input is high*)
		ELSIF
			BitInToCheck AND
			CheckSignalLow AND
			NOT CheckSignalHigh THEN
			TimerTimeOut(Start := TRUE, MTime := (sInit.MaxTime));
			State:=STATE_RUN;
		(* Check input high *)
		ELSIF
			BitInToCheck AND
			NOT CheckSignalLow AND
			CheckSignalHigh THEN
			TimerTimeOut(Start := FALSE, MTime := (sInit.MaxTime));
			State:=State_OK;

		(* Check signal high and input is low*)
		ELSIF
			NOT  BitInToCheck AND
			NOT CheckSignalLow AND
			CheckSignalHigh	THEN
			TimerTimeOut(Start := TRUE, MTime := (sInit.MaxTime));
			State:=STATE_RUN;
		ELSE
			TimerTimeOut(Start := FALSE, MTime := (sInit.MaxTime));

			IF	NOT CheckSignalHigh AND
				NOT CheckSignalLow THEN
				State:=STATE_WAIT;
			END_IF
		END_IF

		(* Timeout check high *)
		IF	TimerTimeOut.Timeout AND
			NOT ResetIntern AND
			State=STATE_RUN AND
			NOT CheckSignalLow AND
			CheckSignalHigh THEN

			State:=STATE_ERROR;
			FB_ReadXmlLineMsg.ID:='SensorFaultNotHigh';

			TempErrorText:=sInit.BitInName;
			TempErrorText:=CONCAT(TempErrorText,' :');
			TempErrorText:=CONCAT(TempErrorText,sVisu.Description);
      			TempErrorText:=CONCAT(TempErrorText,' -> ');
			TempErrorText:=CONCAT(TempErrorText,FB_ReadXmlLineMsg.Text);
			Error.No:=3;
		END_IF
		(* Timeout check low *)
		IF	TimerTimeOut.Timeout AND
			NOT ResetIntern AND
			State=STATE_RUN AND
			CheckSignalLow AND
			NOT CheckSignalHigh THEN
			State:=STATE_ERROR;
			FB_ReadXmlLineMsg.ID:='SensorFaultNotLow';

			TempErrorText:=sInit.BitInName;
			TempErrorText:=CONCAT(TempErrorText,' :');
			TempErrorText:=CONCAT(TempErrorText,sVisu.Description);
      		TempErrorText:=CONCAT(TempErrorText,' -> ');
			TempErrorText:=CONCAT(TempErrorText,FB_ReadXmlLineMsg.Text);
			Error.No:=4;
		END_IF

	ELSE	(* No action *)
		(* Reset ok signal*)
		IF 	State = State_OK AND
			StateOK_CycleFlag THEN
			State:=STATE_WAIT;
		END_IF

	END_IF

END_IF	(* Init ok *)

(*--------------------------------------------------------------------
	Updating processtime (if State_RUN, STATE_ERROR, STATE_RESETS, or STATE_STOPPED)
--------------------------------------------------------------------*)
IF	(State=State_RUN OR
	State=STATE_ERROR OR
	State=STATE_RESETS OR
	State=STATE_STOPPED) AND
	sInit.MaxTime<>0 THEN
	TimerTimeout;
	ProcessTime:=TimerTimeout.PTime;
END_IF

(*------------------------------------------------------------------
	Reset-Handling
  ------------------------------------------------------------------*)
ResetIntern:= 	Reset OR
				BtnReset.Pressed OR
			 	(	State = STATE_ERROR AND
					NOT CheckSignalLow AND
					CheckSignalHigh AND
					BitInToCheck ) OR

			 	(	State = STATE_ERROR AND
					CheckSignalLow AND
					NOT CheckSignalHigh AND
					NOT BitInToCheck) OR

			 	(	State = STATE_ERROR AND
					NOT CheckSignalLow AND
					NOT CheckSignalHigh);

IF 	ResetIntern THEN
	TimerTimeout (Start := FALSE, MTime := (sInit.MaxTime));
	State:= STATE_RESETS;
ELSE
	IF 	State=STATE_RESETS THEN
		State:=STATE_WAIT;
	END_IF
END_IF

(*------------------------------------------------------------------
	Clear all input variables
  ------------------------------------------------------------------*)
Reset:= FALSE;
CheckSignalLow:= FALSE;
CheckSignalHigh:= FALSE;

(*------------------------------------------------------------------
	HomePosition
  ------------------------------------------------------------------*)
HomePositionInfo:=State_OK;

(* Check input signal *)
IF	sInit.HomePosSignal=0 AND
	BitInToCheck THEN
	HomePositionInfo:=11;
END_IF
IF	sInit.HomePosSignal=1 AND
	NOT BitInToCheck THEN
	HomePositionInfo:=10;
END_IF

(* Generating home position*)
(* Zuweisung der Grundstellung*)
IF 	HomePositionInfo=State_OK THEN
	HomePosition:= TRUE;
ELSE
	HomePosition:= FALSE;
	ListHomeNOK(InstName:=sVisu.InstName,Description:=sVisu.Description);
END_IF

(* Objekt-Grundstellung verknüpfen mit GesamtGrundstellung *)
(* object-homeposition concat with mainhomeposition *)
gHomeOk:=gHomeOk AND HomePosition;

(*------------------------------------------------------------------
	Set Visu-Vars
  ------------------------------------------------------------------*)
sVisu.BitInName				:=	sInit.BitInName;
sVisu.BitInToCheck			:=	BitInToCheck;
sVisu.State					:=	State;
sVisu.HomePosition			:=	HomePosition;


(*Copy input-signal to output-var*)
SignalIn:=BitInToCheck;


	(* -------------------------------------------------------------- *)
	(* ------------------ Handle Delay Output --------- *)
	(* -------------------------------------------------------------- *)

	IputOnDelayTime 	(IN := BitInToCheck, PT := DINT_TO_TIME(sInit.IputOnDelayTime));
	IputOffDelayTime 	(IN := BitInToCheck, PT := DINT_TO_TIME(sInit.IputOffDelayTime));

	SignalInDelayed	:=  IputOnDelayTime.Q  OR (IputOffDelayTime.Q AND NOT BitInToCheck);

(*------------------------------------------------------------------
	Error-Handling
  ------------------------------------------------------------------*)
	LaufschriftObj(
	N:= 40,
	StepWidth:=1,
	PT:= t#100ms ,
	Text:= TempErrorText,
	Display=>sVisu.ErrorString );

	LaufschriftErrh(
	N:= 160,
	StepWidth:=1,
	PT:= t#100ms ,
	Text:= TempErrorText,
	Display=>Error.Text );

(*  *)
IF State=STATE_ERROR AND
	NOT ErrorElapsed THEN
	ErrorElapsed:=TRUE;
	Error.DateTime:=gVarDTSystemtime;
END_IF

IF 	State<>STATE_ERROR THEN
	ErrorElapsed:=FALSE;
	TempErrorText:='';
END_IF;

sVisu.ProcessTime:=ProcessTime;

IF 	Error.Text<>''	AND ST_Lng.b_EndChangeLng THEN
	Error.Typ:=0;
	ErrorHandler.AddError(ErrorToAdd:=Error,
	sVisu:=Visu.ErrorHandler);
END_IF

(* ------------------------------------------------------------------------------------------ *)
(* ---------------- LANGUAGE auslesen aus der XML Datei-------- *)
(* ------------------------------------------------------------------------------------------ *)
sVisu.BitInName:=sInit.BitInName;
sVisu.InstName:=sInit.InstName;
sVisu.ErrorPresent:=Error.Text<>'';

FB_ReadXmlLineConf(
	Prefix:= 'CONFIG',
	ID:= sInit.InstName,
	File:= 'CONFIG.xml',
	Text=> sVisu.Description  );


FB_ReadXmlLineMsg(
	Prefix:= 'MSG',
	ID:= ,
	File:= 'MSG.xml',
	Text=>);

IF 	State = STATE_ERROR THEN
	TempErrorText:=sInit.BitInName;
	TempErrorText:=CONCAT(TempErrorText,' :');
	TempErrorText:=CONCAT(TempErrorText,sVisu.Description);
	TempErrorText:=CONCAT(TempErrorText,' -> ');
	TempErrorText:=CONCAT(TempErrorText,FB_ReadXmlLineMsg.Text);
END_IF
END_FUNCTION_BLOCK

(* POU zLibrary/DigOutIn/FB_DigOutIn, ST *)
FUNCTION_BLOCK FB_DigOutIn (*Version 1.2, 20.NOV 2010*)
VAR_OUTPUT
	State					: StateObject;	(* State of the object *)
	HomePosition			: BOOL;					(* object in home-position*)
	SignalOut				: BOOL;							(* Static signal of digital output *)
	SignalIn				: BOOL;							(* Static signal of digital input *)
END_VAR
VAR_INPUT
	SetSignalHigh			: BOOL;		 		 	(* Signal set  HIGH *)
	SetSignalLow			: BOOL;		 			(* Signal set  LOW  *)

	PulseOn					: BOOL;		 			(* Signal pulse On *)
	PulseTime				: DINT; 				(* Length in ms for output impulse *)

	FlashSignal				: BOOL;		 			(* Signal FLASH  *)
	OnTime					: DINT; 				(* In ms for ON time *)
	OffTime					: DINT; 				(* In ms for OFF time *)

	CheckSignalHigh			: BOOL;		 		 	(* Signal check  HIGH *)
	CheckSignalLow			: BOOL;		 			(* Signal check  LOW  *)

	Enable					: BOOL:=TRUE; 	(* Enables the operations on the class *)
	Reset					: BOOL;					(* switch for resetting the control *)

	SFCCurrentStep			: STRING(40);		(* aktually step in the order of events *)
	SFCCurrentPOU			: STRING(40);		(* Name of the order of events*)

	sInit					: sDigOutInInit;		(* Initializingvalues to the Instance *)
	strAnlayse				: STRING(255);  (*String to analyse Lockings*)
END_VAR
VAR_IN_OUT
	sVisu					: sDigOutInVisu;
END_VAR
VAR
	BitOutToSet				AT %Q* :BOOL;		(* Bit output signal to set *)
	BitInToCheck			AT %I* :BOOL;		(* Bit input signal to check *)

	ProcessTime				: DINT;					(* Counts the time in steps of 100ms since starting operation *)

	TimerTimeOut			: CheckProcTime;		(* Timer generates timeout signal *)
	Error					: ErrorStruct;
	ErrorElapsed			: R_TRIG;
	LaufschriftErrh			: FB_Laufschrift;
	LaufschriftObj			: FB_Laufschrift_STR255;
	LaufschriftAnalyse		: FB_Laufschrift_STR255;
	TempString				: STRING(255);

	TempErrorText			: STRING(255);
	OutputAvailable			: BOOL;
	InputAvailable			: BOOL;
	HomePositionInfo		: DINT;							(* missing to home posistion *)
	ResetIntern				: BOOL;							(* Internal reset signal *)
	InitState				: BOOL :=FALSE;		(* Internal State for initialising *)

	BtnOutput				: VisuButton;			(* Manage button *)
	BtnReset				: VisuButton;			(* Manage button *)

	SetOutPulse				: TP;							(* Timer for set output pulse *)
	SetOutPulseActive		: BOOL;
	TimerOn		 			: TON;						(* Timer for output on time *)
	TimerOff		 		: TOF;						(* Timer for output off time *)
  	StateOK_CycleFlag		: BOOL;

	FB_ReadXmlLineConf		: FB_ReadXmlLine;
	FB_ReadXmlLineMsg		: FB_ReadXmlLine;

END_VAR
VAR CONSTANT
	INPUT_CHECKLOW			: DINT:=  21;	(* State input check low *)
	INPUT_CHECKHIGH			: DINT:=  22;	(* State input check  high *)
END_VAR
Error.No:=0;
Error.Text:='';

(*------------------------------------------------------------------
	Initialization
  ------------------------------------------------------------------*)
IF 	NOT InitState THEN
	InitState:=TRUE;

	(* Check instance name *)
	IF 	sInit.InstName='' THEN
		InitState:=FALSE;
		State:=STATE_ERROR;
		Error.No:=4;
		TempErrorText:='InstName not defined';

	(* Check input name *)
	ELSIF
		sInit.BitOutName='' AND  sInit.BitInName='' THEN

		InitState:=FALSE;
		State:=STATE_ERROR;
		Error.No:=4;
		TempErrorText:='No bit out and in name defined';
		sInit.BitOutName:='No output name!';
		sInit.BitInName:='No input name!';
	END_IF

	(* Check output name *)
	IF 	sInit.BitOutName<>'' THEN
		OutputAvailable:=TRUE;
	ELSE
		OutputAvailable:=FALSE;
		sInit.BitOutName:='No output name!';
	END_IF

	(* Check input name *)
	IF 	sInit.BitInName<>'' 	THEN
		InputAvailable:=TRUE;
	ELSE
		InputAvailable:=FALSE;
		sInit.BitInName:='No input name!';
	END_IF

	(* send names to Visu *)
	sVisu.InstName	:= sInit.InstName;
	sVisu.Description	:= sInit.Description;
	sVisu.BitOutName	:= sInit.BitOutName;
	sVisu.InputAvailable	:= InputAvailable;
	sVisu.OutputAvailable	:= OutputAvailable;

END_IF

(* Add InitState to Global-Init-State to collect all Objects *)
gInitCollect:=gInitCollect AND InitState;

IF gInitOk THEN
StateOK_CycleFlag := NOT (State<>State_ok);

(*------------------------------------------------------------------
	Show and Read Buttons
  ------------------------------------------------------------------*)
	BtnOutput(Button:=sVisu.BtnOutput,
						Enable:=(ModeSelect.Mode=MODE_MANUAL OR sInit.EnableVisuInEveryMode ) AND Enable AND OutputAvailable  ,
						Visible:= OutputAvailable,
						TextOn:=sInit.BitOutName,
						TextOff:=sInit.BitOutName,
						PressedExt:=FALSE ,
						StateOn:= FALSE ,
						);

	(*------------------------------------------------------------------
	Manual-Mode
  ------------------------------------------------------------------*)
	IF  	ModeSelect.Mode=MODE_MANUAL OR
		sInit.EnableVisuInEveryMode THEN
		(* Set or reset output manual *)
		IF	BtnOutput.PressedFlag AND
			OutputAvailable AND
			Enable	THEN
			IF 	NOT BitOutToSet THEN
				BitOutToSet:=TRUE;
			ELSE
				BitOutToSet:=FALSE;
			END_IF
		END_IF

		SFCCurrentStep:=sInit.InstName;
		SFCCurrentPOU:='MODE_MANUAL';
	END_IF (*ModeSelect.Mode=MODE_MANUAL*)

	(*------------------------------------------------------------------
	Mode higher manual mode (auto, tip or homeposrun)
  ------------------------------------------------------------------*)
	IF 		(ModeSelect.Mode>MODE_MANUAL OR sInit.EnableInEveryMode OR sInit.EnableVisuInEveryMode) AND
			(	SetSignalHigh OR
				 SetSignalLow OR
				 PulseOn OR
				 SetOutPulseActive OR
				 FlashSignal OR
				 CheckSignalHigh OR
				 CheckSignalLow 	) THEN
	
		(* Set output on off                                       *)
		(*=========================================================*)

		(* Set output signal *)
		IF	SetSignalHigh AND
			NOT SetSignalLow AND
			NOT PulseOn AND
			NOT FlashSignal AND
			OutputAvailable THEN

			BitOutToSet:=TRUE;

			(* If no sensor check then state ok *)
			IF 	NOT InputAvailable	OR
				( NOT CheckSignalHigh AND
				  NOT CheckSignalLow )	THEN

				State:=STATE_OK;
			END_IF
		END_IF
		
		(* Reset output signal *)
		IF	NOT SetSignalHigh AND
			SetSignalLow AND
			NOT PulseOn AND
			NOT FlashSignal AND
			OutputAvailable 	THEN

			BitOutToSet:=FALSE;

			(* If no sensor check then state ok *)
			IF 	NOT InputAvailable OR
				( NOT CheckSignalHigh AND
				  NOT CheckSignalLow )	THEN

				State:=STATE_OK;
			END_IF
		END_IF

		(* Set output with pulse time                              *)
		(*=========================================================*)
		IF	PulseOn OR SetOutPulseActive AND
			OutputAvailable AND
			PulseTime>0 AND
			NOT SetSignalHigh AND
			NOT SetSignalLow AND
			NOT FlashSignal THEN

			SetOutPulse(IN:=TRUE,	PT:=DINT_TO_TIME(PulseTime)	);

			BitOutToSet:=SetOutPulse.Q;
			SetOutPulseActive:=TRUE;
			(* Pulse finished *)
			IF	NOT SetOutPulse.Q	THEN
				SetOutPulse(IN:=FALSE, PT:=T#0s);
				SetOutPulseActive:=FALSE;
			(* If no sensor check then state ok *)
			IF	NOT	InputAvailable OR
				(NOT CheckSignalHigh AND
				 NOT CheckSignalLow) THEN

				State:=STATE_OK;
				END_IF
			END_IF
		END_IF


		(* Set output with on and off time                         *)
		(*=========================================================*)
		IF	FlashSignal AND
			OnTime>0 AND
			OffTime>0 AND
			OutputAvailable AND

			NOT PulseOn AND
			NOT SetSignalHigh AND
			NOT SetSignalLow THEN

			TimerOn(IN:=TimerOff.Q = FALSE , PT:=DINT_TO_TIME(OnTime)); (* On time *)
			TimerOff(IN:=TimerOn.Q = TRUE, PT:=DINT_TO_TIME(OffTime));	(* Off time *)

			(* assign output *)
			IF 	NOT TimerOff.Q THEN
				BitOutToSet:=TRUE;
			ELSE
				BitOutToSet:=FALSE;
			END_IF

			(* If no sensor check then state ok *)
			IF 	NOT InputAvailable OR
				(NOT CheckSignalHigh AND
				 NOT CheckSignalLow) THEN

				State:=STATE_OK;
			END_IF
		
		
		END_IF
	
	
	(* Check input signal                                      *)
	(*=========================================================*)
	
		(* Check signal low and input is low*)
		IF	NOT 	BitInToCheck AND
			InputAvailable AND
			CheckSignalLow AND
			NOT CheckSignalHigh THEN

			(* Check input low and it is low *)
			TimerTimeOut(Start := FALSE, MTime := (sInit.MaxTime));
			State:=State_OK;

		(* Check input low and input is high*)
		ELSIF
			BitInToCheck AND
			InputAvailable AND
			CheckSignalLow AND
			NOT CheckSignalHigh THEN

			TimerTimeOut(Start := TRUE, MTime := (sInit.MaxTime));
			State:=STATE_ERROR (*INPUT_CHECKLOW*);
			FB_ReadXmlLineMsg.ID:='SensorFaultNotLow';

			TempErrorText:=sVisu.InstName;
			TempErrorText:=CONCAT(TempErrorText,' ');
			TempErrorText:=CONCAT(TempErrorText,sVisu.Description);
			TempErrorText:=CONCAT(TempErrorText,'  ');
			TempErrorText:=CONCAT(TempErrorText,FB_ReadXmlLineMsg.Text);

			Error.No:=1;

